LIN {X 0,Y 511.911,Z 787.73,A -85,B 0,C 180,E1 -4052.8,E2 -4052.8} C_VEL
LIN {X 0,Y 511.92,Z 784.945,A -85,B 0,C 180,E1 -4055.058,E2 -4055.058} C_VEL
LIN {X 0,Y 511.96,Z 780.479,A -85,B 0,C 180,E1 -4057.294,E2 -4057.294} C_VEL
LIN {X 0,Y 512.078,Z 774.263,A -85,B 0,C 180,E1 -4059.555,E2 -4059.555} C_VEL
LIN {X 0,Y 512.293,Z 766.172,A -85,B 0,C 180,E1 -4061.827,E2 -4061.827} C_VEL
LIN {X 0,Y 512.637,Z 756.556,A -85,B 0,C 180,E1 -4063.997,E2 -4063.997} C_VEL
LIN {X 0,Y 513.141,Z 745.479,A -85,B 0,C 180,E1 -4066.064,E2 -4066.064} C_VEL
LIN {X 0,Y 513.792,Z 732.943,A -85,B 0,C 180,E1 -4068.025,E2 -4068.025} C_VEL
LIN {X 0,Y 514.601,Z 718.86,A -85,B 0,C 180,E1 -4069.881,E2 -4069.881} C_VEL
LIN {X 0,Y 515.516,Z 703.77,A -85,B 0,C 180,E1 -4071.571,E2 -4071.571} C_VEL
LIN {X 0,Y 516.554,Z 687.043,A -85,B 0,C 180,E1 -4073.158,E2 -4073.158} C_VEL
LIN {X 0,Y 517.654,Z 668.921,A -85,B 0,C 180,E1 -4074.599,E2 -4074.599} C_VEL
LIN {X 0,Y 518.736,Z 650.255,A -85,B 0,C 180,E1 -4075.825,E2 -4075.825} C_VEL
LIN {X 0,Y 519.635,Z 632.605,A -85,B 0,C 180,E1 -4076.772,E2 -4076.772} C_VEL
LIN {X 0,Y 520.342,Z 613.516,A -85,B 0,C 180,E1 -4077.557,E2 -4077.557} C_VEL
LIN {X 0,Y 520.963,Z 593.158,A -85,B 0,C 180,E1 -4078.186,E2 -4078.186} C_VEL
LIN {X 0,Y 521.396,Z 571.634,A -85,B 0,C 180,E1 -4078.64,E2 -4078.64} C_VEL
LIN {X 0,Y 522.992,Z 374.414,A -85,B 0,C 180,E1 -4081.484,E2 -4081.484} C_VEL
LIN {X 0,Y 523.224,Z 329.363,A -85,B 0,C 180,E1 -4082.176,E2 -4082.176} C_VEL
LIN {X 0,Y 521.156,Z 316.493,A -85,B 0,C 180,E1 -4082.526,E2 -4082.526} C_VEL
LIN {X 0,Y 521.816,Z 297.274,A -85,B 0,C 180,E1 -4083.935,E2 -4083.935} C_VEL
LIN {X 0,Y 514.978,Z 278.961,A -85,B 0,C 180,E1 -4085.941,E2 -4085.941} C_VEL
LIN {X 0,Y 512.679,Z 272.854,A -85,B 0,C 180,E1 -4086.732,E2 -4086.732} C_VEL
LIN {X 0,Y 512.623,Z 272.631,A -85,B 0,C 180,E1 -4090.13,E2 -4090.13} C_VEL
LIN {X 0,Y 512.61,Z 272.633,A -85,B 0,C 180,E1 -4093.67,E2 -4093.67} C_VEL
LIN {X 0,Y 512.639,Z 272.631,A -85,B 0,C 180,E1 -4097.102,E2 -4097.102} C_VEL
LIN {X 0,Y 512.649,Z 272.63,A -85,B 0,C 180,E1 -4100.566,E2 -4100.566} C_VEL
LIN {X 0,Y 512.604,Z 272.635,A -85,B 0,C 180,E1 -4103.91,E2 -4103.91} C_VEL
LIN {X 0,Y 512.644,Z 272.869,A -85,B 0,C 180,E1 -4105.454,E2 -4105.454} C_VEL
LIN {X 0,Y 516.614,Z 283.424,A -85,B 0,C 180,E1 -4106.934,E2 -4106.934} C_VEL
LIN {X 0,Y 520.776,Z 295.802,A -85,B 0,C 180,E1 -4108.454,E2 -4108.454} C_VEL
LIN {X 0,Y 518.7,Z 337.157,A -85,B 0,C 180,E1 -4112.069,E2 -4112.069} C_VEL
LIN {X 0,Y 518.616,Z 342.587,A -85,B 0,C 180,E1 -4112.489,E2 -4112.489} C_VEL
LIN {X 0,Y 520.868,Z 357.617,A -85,B 0,C 180,E1 -4112.895,E2 -4112.895} C_VEL
LIN {X 0,Y 518.908,Z 559.958,A -85,B 0,C 180,E1 -4115.886,E2 -4115.886} C_VEL
LIN {X 0,Y 518.407,Z 579.62,A -85,B 0,C 180,E1 -4116.386,E2 -4116.386} C_VEL
LIN {X 0,Y 517.798,Z 597.604,A -85,B 0,C 180,E1 -4117.042,E2 -4117.042} C_VEL
LIN {X 0,Y 517.068,Z 615.514,A -85,B 0,C 180,E1 -4117.908,E2 -4117.908} C_VEL
LIN {X 0,Y 516.22,Z 633.368,A -85,B 0,C 180,E1 -4119.003,E2 -4119.003} C_VEL
LIN {X 0,Y 515.38,Z 650.152,A -85,B 0,C 180,E1 -4120.272,E2 -4120.272} C_VEL
LIN {X 0,Y 514.552,Z 665.731,A -85,B 0,C 180,E1 -4121.711,E2 -4121.711} C_VEL
LIN {X 0,Y 513.83,Z 679.746,A -85,B 0,C 180,E1 -4123.263,E2 -4123.263} C_VEL
LIN {X 0,Y 513.204,Z 692.76,A -85,B 0,C 180,E1 -4124.983,E2 -4124.983} C_VEL
LIN {X 0,Y 512.71,Z 704.206,A -85,B 0,C 180,E1 -4126.811,E2 -4126.811} C_VEL
LIN {X 0,Y 512.352,Z 714.139,A -85,B 0,C 180,E1 -4128.747,E2 -4128.747} C_VEL
LIN {X 0,Y 512.116,Z 722.573,A -85,B 0,C 180,E1 -4130.788,E2 -4130.788} C_VEL
LIN {X 0,Y 511.992,Z 729.132,A -85,B 0,C 180,E1 -4132.821,E2 -4132.821} C_VEL
LIN {X 0,Y 511.937,Z 734.158,A -85,B 0,C 180,E1 -4134.958,E2 -4134.958} C_VEL
LIN {X 0,Y 511.914,Z 737.334,A -85,B 0,C 180,E1 -4137.09,E2 -4137.09} C_VEL
LIN {X 0,Y 511.917,Z 738.827,A -85,B 0,C 180,E1 -4139.217,E2 -4139.217} C_VEL
LIN {X 0,Y 511.911,Z 738.673,A -85,B 0,C 180,E1 -4141.343,E2 -4141.343} C_VEL
LIN {X 0,Y 511.912,Z 736.707,A -85,B 0,C 180,E1 -4143.547,E2 -4143.547} C_VEL
LIN {X 0,Y 511.942,Z 732.933,A -85,B 0,C 180,E1 -4145.717,E2 -4145.717} C_VEL
LIN {X 0,Y 512.015,Z 727.399,A -85,B 0,C 180,E1 -4147.857,E2 -4147.857} C_VEL
LIN {X 0,Y 512.174,Z 720.364,A -85,B 0,C 180,E1 -4149.892,E2 -4149.892} C_VEL
LIN {X 0,Y 512.432,Z 711.904,A -85,B 0,C 180,E1 -4151.823,E2 -4151.823} C_VEL
LIN {X 0,Y 512.822,Z 701.375,A -85,B 0,C 180,E1 -4153.761,E2 -4153.761} C_VEL
LIN {X 0,Y 513.355,Z 689.287,A -85,B 0,C 180,E1 -4155.592,E2 -4155.592} C_VEL
LIN {X 0,Y 514.033,Z 675.591,A -85,B 0,C 180,E1 -4157.314,E2 -4157.314} C_VEL
LIN {X 0,Y 514.776,Z 661.344,A -85,B 0,C 180,E1 -4158.81,E2 -4158.81} C_VEL
LIN {X 0,Y 515.609,Z 645.529,A -85,B 0,C 180,E1 -4160.193,E2 -4160.193} C_VEL
LIN {X 0,Y 516.449,Z 628.721,A -85,B 0,C 180,E1 -4161.398,E2 -4161.398} C_VEL
LIN {X 0,Y 517.278,Z 610.536,A -85,B 0,C 180,E1 -4162.443,E2 -4162.443} C_VEL
LIN {X 0,Y 518.022,Z 591.934,A -85,B 0,C 180,E1 -4163.277,E2 -4163.277} C_VEL
LIN {X 0,Y 518.599,Z 572.89,A -85,B 0,C 180,E1 -4163.901,E2 -4163.901} C_VEL
LIN {X 0,Y 519.014,Z 553.054,A -85,B 0,C 180,E1 -4164.326,E2 -4164.326} C_VEL
LIN {X 0,Y 520.123,Z 426.027,A -85,B 0,C 180,E1 -4166.177,E2 -4166.177} C_VEL
LIN {X 0,Y 519.314,Z 418.442,A -85,B 0,C 180,E1 -4166.337,E2 -4166.337} C_VEL
LIN {X 0,Y 513.976,Z 398.623,A -85,B 0,C 180,E1 -4166.947,E2 -4166.947} C_VEL
LIN {X 0,Y 513.364,Z 392.104,A -85,B 0,C 180,E1 -4167.084,E2 -4167.084} C_VEL
LIN {X 0,Y 513.545,Z 356.301,A -85,B 0,C 180,E1 -4167.633,E2 -4167.633} C_VEL
LIN {X 0,Y 511.161,Z 341.819,A -85,B 0,C 180,E1 -4168.047,E2 -4168.047} C_VEL
LIN {X 0,Y 513.119,Z 299.865,A -85,B 0,C 180,E1 -4171.679,E2 -4171.679} C_VEL
LIN {X 0,Y 513.068,Z 297.719,A -85,B 0,C 180,E1 -4171.879,E2 -4171.879} C_VEL
LIN {X 0,Y 506.338,Z 278.626,A -85,B 0,C 180,E1 -4174.167,E2 -4174.167} C_VEL
LIN {X 0,Y 504.722,Z 273.804,A -85,B 0,C 180,E1 -4174.805,E2 -4174.805} C_VEL
LIN {X 0,Y 504.673,Z 273.62,A -85,B 0,C 180,E1 -4178.181,E2 -4178.181} C_VEL
LIN {X 0,Y 504.694,Z 273.612,A -85,B 0,C 180,E1 -4181.678,E2 -4181.678} C_VEL
LIN {X 0,Y 504.706,Z 273.617,A -85,B 0,C 180,E1 -4185.173,E2 -4185.173} C_VEL
LIN {X 0,Y 504.71,Z 273.619,A -85,B 0,C 180,E1 -4188.723,E2 -4188.723} C_VEL
LIN {X 0,Y 504.699,Z 273.618,A -85,B 0,C 180,E1 -4192.253,E2 -4192.253} C_VEL
LIN {X 0,Y 504.707,Z 273.613,A -85,B 0,C 180,E1 -4195.762,E2 -4195.762} C_VEL
LIN {X 0,Y 504.69,Z 273.612,A -85,B 0,C 180,E1 -4199.297,E2 -4199.297} C_VEL
LIN {X 0,Y 504.681,Z 273.619,A -85,B 0,C 180,E1 -4202.817,E2 -4202.817} C_VEL
LIN {X 0,Y 504.705,Z 273.616,A -85,B 0,C 180,E1 -4206.286,E2 -4206.286} C_VEL
LIN {X 0,Y 504.708,Z 273.614,A -85,B 0,C 180,E1 -4209.835,E2 -4209.835} C_VEL
LIN {X 0,Y 504.659,Z 273.622,A -85,B 0,C 180,E1 -4213.185,E2 -4213.185} C_VEL
LIN {X 0,Y 504.648,Z 273.601,A -85,B 0,C 180,E1 -4216.712,E2 -4216.712} C_VEL
LIN {X 0,Y 504.657,Z 273.717,A -85,B 0,C 180,E1 -4219.208,E2 -4219.208} C_VEL
LIN {X 0,Y 505.095,Z 275.399,A -85,B 0,C 180,E1 -4219.448,E2 -4219.448} C_VEL
LIN {X 0,Y 511.329,Z 294.509,A -85,B 0,C 180,E1 -4221.424,E2 -4221.424} C_VEL
LIN {X 0,Y 510.714,Z 334.383,A -85,B 0,C 180,E1 -4224.663,E2 -4224.663} C_VEL
LIN {X 0,Y 509.833,Z 376.612,A -85,B 0,C 180,E1 -4228.088,E2 -4228.088} C_VEL
LIN {X 0,Y 508.721,Z 421.729,A -85,B 0,C 180,E1 -4231.744,E2 -4231.744} C_VEL
LIN {X 0,Y 507.706,Z 464.389,A -85,B 0,C 180,E1 -4235.196,E2 -4235.196} C_VEL
LIN {X 0,Y 507.513,Z 474.435,A -85,B 0,C 180,E1 -4235.982,E2 -4235.982} C_VEL
LIN {X 0,Y 508.534,Z 485.17,A -85,B 0,C 180,E1 -4236.182,E2 -4236.182} C_VEL
LIN {X 0,Y 507.591,Z 616.922,A -85,B 0,C 180,E1 -4238.102,E2 -4238.102} C_VEL
LIN {X 0,Y 507.323,Z 632.874,A -85,B 0,C 180,E1 -4238.542,E2 -4238.542} C_VEL
LIN {X 0,Y 506.925,Z 648.572,A -85,B 0,C 180,E1 -4239.192,E2 -4239.192} C_VEL
LIN {X 0,Y 506.455,Z 663.014,A -85,B 0,C 180,E1 -4240.003,E2 -4240.003} C_VEL
LIN {X 0,Y 505.905,Z 677.326,A -85,B 0,C 180,E1 -4241.051,E2 -4241.051} C_VEL
LIN {X 0,Y 505.414,Z 690.119,A -85,B 0,C 180,E1 -4242.234,E2 -4242.234} C_VEL
LIN {X 0,Y 504.93,Z 702.107,A -85,B 0,C 180,E1 -4243.628,E2 -4243.628} C_VEL
LIN {X 0,Y 504.569,Z 711.921,A -85,B 0,C 180,E1 -4245.044,E2 -4245.044} C_VEL
LIN {X 0,Y 504.268,Z 721.08,A -85,B 0,C 180,E1 -4246.724,E2 -4246.724} C_VEL
LIN {X 0,Y 504.091,Z 728.094,A -85,B 0,C 180,E1 -4248.382,E2 -4248.382} C_VEL
LIN {X 0,Y 503.989,Z 733.734,A -85,B 0,C 180,E1 -4250.217,E2 -4250.217} C_VEL
LIN {X 0,Y 503.95,Z 737.461,A -85,B 0,C 180,E1 -4252.022,E2 -4252.022} C_VEL
LIN {X 0,Y 503.935,Z 739.424,A -85,B 0,C 180,E1 -4253.874,E2 -4253.874} C_VEL
LIN {X 0,Y 503.935,Z 739.676,A -85,B 0,C 180,E1 -4255.753,E2 -4255.753} C_VEL
LIN {X 0,Y 503.943,Z 738.029,A -85,B 0,C 180,E1 -4257.661,E2 -4257.661} C_VEL
LIN {X 0,Y 503.976,Z 734.754,A -85,B 0,C 180,E1 -4259.471,E2 -4259.471} C_VEL
LIN {X 0,Y 504.057,Z 729.721,A -85,B 0,C 180,E1 -4261.246,E2 -4261.246} C_VEL
LIN {X 0,Y 504.23,Z 722.652,A -85,B 0,C 180,E1 -4263.044,E2 -4263.044} C_VEL
LIN {X 0,Y 504.492,Z 714.234,A -85,B 0,C 180,E1 -4264.665,E2 -4264.665} C_VEL
LIN {X 0,Y 504.853,Z 704.388,A -85,B 0,C 180,E1 -4266.168,E2 -4266.168} C_VEL
LIN {X 0,Y 505.3,Z 693.074,A -85,B 0,C 180,E1 -4267.548,E2 -4267.548} C_VEL
LIN {X 0,Y 505.831,Z 679.711,A -85,B 0,C 180,E1 -4268.848,E2 -4268.848} C_VEL
LIN {X 0,Y 506.327,Z 666.781,A -85,B 0,C 180,E1 -4269.842,E2 -4269.842} C_VEL
LIN {X 0,Y 506.852,Z 651.387,A -85,B 0,C 180,E1 -4270.763,E2 -4270.763} C_VEL
LIN {X 0,Y 507.266,Z 635.918,A -85,B 0,C 180,E1 -4271.442,E2 -4271.442} C_VEL
LIN {X 0,Y 507.556,Z 619.27,A -85,B 0,C 180,E1 -4271.94,E2 -4271.94} C_VEL
LIN {X 0,Y 507.753,Z 593.359,A -85,B 0,C 180,E1 -4272.356,E2 -4272.356} C_VEL
LIN {X 0,Y 508.34,Z 481.293,A -85,B 0,C 180,E1 -4273.974,E2 -4273.974} C_VEL
LIN {X 0,Y 507.457,Z 474.005,A -85,B 0,C 180,E1 -4274.135,E2 -4274.135} C_VEL
LIN {X 0,Y 508.502,Z 429.195,A -85,B 0,C 180,E1 -4277.741,E2 -4277.741} C_VEL
LIN {X 0,Y 509.471,Z 389.356,A -85,B 0,C 180,E1 -4280.951,E2 -4280.951} C_VEL
LIN {X 0,Y 510.24,Z 346.659,A -85,B 0,C 180,E1 -4284.346,E2 -4284.346} C_VEL
LIN {X 0,Y 510.701,Z 309.068,A -85,B 0,C 180,E1 -4287.334,E2 -4287.334} C_VEL
LIN {X 0,Y 510.741,Z 292.979,A -85,B 0,C 180,E1 -4288.618,E2 -4288.618} C_VEL
LIN {X 0,Y 504.771,Z 274.004,A -85,B 0,C 180,E1 -4290.512,E2 -4290.512} C_VEL
LIN {X 0,Y 504.69,Z 273.619,A -85,B 0,C 180,E1 -4290.885,E2 -4290.885} C_VEL
LIN {X 0,Y 504.709,Z 273.616,A -85,B 0,C 180,E1 -4294.336,E2 -4294.336} C_VEL
LIN {X 0,Y 504.669,Z 273.622,A -85,B 0,C 180,E1 -4297.764,E2 -4297.764} C_VEL
LIN {X 0,Y 504.671,Z 273.614,A -85,B 0,C 180,E1 -4301.279,E2 -4301.279} C_VEL
LIN {X 0,Y 504.711,Z 273.613,A -85,B 0,C 180,E1 -4304.739,E2 -4304.739} C_VEL
LIN {X 0,Y 504.694,Z 273.622,A -85,B 0,C 180,E1 -4308.225,E2 -4308.225} C_VEL
LIN {X 0,Y 504.667,Z 273.617,A -85,B 0,C 180,E1 -4311.684,E2 -4311.684} C_VEL
LIN {X 0,Y 504.687,Z 273.615,A -85,B 0,C 180,E1 -4315.192,E2 -4315.192} C_VEL
LIN {X 0,Y 504.711,Z 273.617,A -85,B 0,C 180,E1 -4318.637,E2 -4318.637} C_VEL
LIN {X 0,Y 504.675,Z 273.618,A -85,B 0,C 180,E1 -4322.043,E2 -4322.043} C_VEL
LIN {X 0,Y 504.673,Z 273.617,A -85,B 0,C 180,E1 -4325.571,E2 -4325.571} C_VEL
LIN {X 0,Y 504.709,Z 273.612,A -85,B 0,C 180,E1 -4329.004,E2 -4329.004} C_VEL
LIN {X 0,Y 504.704,Z 273.617,A -85,B 0,C 180,E1 -4332.586,E2 -4332.586} C_VEL
LIN {X 0,Y 504.673,Z 273.615,A -85,B 0,C 180,E1 -4335.985,E2 -4335.985} C_VEL
LIN {X 0,Y 504.69,Z 273.614,A -85,B 0,C 180,E1 -4339.441,E2 -4339.441} C_VEL
LIN {X 0,Y 504.712,Z 273.617,A -85,B 0,C 180,E1 -4342.971,E2 -4342.971} C_VEL
LIN {X 0,Y 504.691,Z 273.62,A -85,B 0,C 180,E1 -4346.471,E2 -4346.471} C_VEL
LIN {X 0,Y 504.676,Z 273.615,A -85,B 0,C 180,E1 -4349.951,E2 -4349.951} C_VEL
LIN {X 0,Y 504.704,Z 273.613,A -85,B 0,C 180,E1 -4353.417,E2 -4353.417} C_VEL
LIN {X 0,Y 504.708,Z 273.62,A -85,B 0,C 180,E1 -4356.888,E2 -4356.888} C_VEL
LIN {X 0,Y 504.68,Z 273.619,A -85,B 0,C 180,E1 -4360.379,E2 -4360.379} C_VEL
LIN {X 0,Y 504.684,Z 273.618,A -85,B 0,C 180,E1 -4363.9,E2 -4363.9} C_VEL
LIN {X 0,Y 504.71,Z 273.617,A -85,B 0,C 180,E1 -4367.352,E2 -4367.352} C_VEL
LIN {X 0,Y 504.713,Z 273.617,A -85,B 0,C 180,E1 -4370.954,E2 -4370.954} C_VEL
LIN {X 0,Y 504.722,Z 273.854,A -85,B 0,C 180,E1 -4372.645,E2 -4372.645} C_VEL
LIN {X 0,Y 507.634,Z 281.444,A -85,B 0,C 180,E1 -4373.571,E2 -4373.571} C_VEL
LIN {X 0,Y 515.207,Z 300.924,A -85,B 0,C 180,E1 -4375.719,E2 -4375.719} C_VEL
LIN {X 0,Y 514.589,Z 316.443,A -85,B 0,C 180,E1 -4376.864,E2 -4376.864} C_VEL
LIN {X 0,Y 517.105,Z 333.218,A -85,B 0,C 180,E1 -4377.321,E2 -4377.321} C_VEL
LIN {X 0,Y 514.727,Z 530.291,A -85,B 0,C 180,E1 -4380.332,E2 -4380.332} C_VEL
LIN {X 0,Y 514.183,Z 578.441,A -85,B 0,C 180,E1 -4381.071,E2 -4381.071} C_VEL
LIN {X 0,Y 513.538,Z 599.827,A -85,B 0,C 180,E1 -4381.608,E2 -4381.608} C_VEL
LIN {X 0,Y 512.738,Z 620.455,A -85,B 0,C 180,E1 -4382.349,E2 -4382.349} C_VEL
LIN {X 0,Y 511.825,Z 639.514,A -85,B 0,C 180,E1 -4383.24,E2 -4383.24} C_VEL
LIN {X 0,Y 510.774,Z 658.935,A -85,B 0,C 180,E1 -4384.368,E2 -4384.368} C_VEL
LIN {X 0,Y 509.701,Z 677.368,A -85,B 0,C 180,E1 -4385.674,E2 -4385.674} C_VEL
LIN {X 0,Y 508.649,Z 693.186,A -85,B 0,C 180,E1 -4387.035,E2 -4387.035} C_VEL
LIN {X 0,Y 507.519,Z 709.709,A -85,B 0,C 180,E1 -4388.725,E2 -4388.725} C_VEL
LIN {X 0,Y 506.541,Z 724.454,A -85,B 0,C 180,E1 -4390.515,E2 -4390.515} C_VEL
LIN {X 0,Y 505.731,Z 737.586,A -85,B 0,C 180,E1 -4392.394,E2 -4392.394} C_VEL
LIN {X 0,Y 505.077,Z 749.383,A -85,B 0,C 180,E1 -4394.383,E2 -4394.383} C_VEL
LIN {X 0,Y 504.568,Z 760.338,A -85,B 0,C 180,E1 -4396.596,E2 -4396.596} C_VEL
LIN {X 0,Y 504.236,Z 769.256,A -85,B 0,C 180,E1 -4398.796,E2 -4398.796} C_VEL
LIN {X 0,Y 504.048,Z 776.587,A -85,B 0,C 180,E1 -4401.062,E2 -4401.062} C_VEL
LIN {X 0,Y 503.957,Z 782.261,A -85,B 0,C 180,E1 -4403.394,E2 -4403.394} C_VEL
LIN {X 0,Y 503.916,Z 786.089,A -85,B 0,C 180,E1 -4405.677,E2 -4405.677} C_VEL
LIN {X 0,Y 503.911,Z 788.374,A -85,B 0,C 180,E1 -4408.068,E2 -4408.068} C_VEL
LIN {X 0,Y 503.9,Z 788.917,A -85,B 0,C 180,E1 -4410.456,E2 -4410.456} C_VEL
LIN {X 0,Y 503.911,Z 787.842,A -85,B 0,C 180,E1 -4412.731,E2 -4412.731} C_VEL
LIN {X 0,Y 503.922,Z 785.126,A -85,B 0,C 180,E1 -4415.01,E2 -4415.01} C_VEL
LIN {X 0,Y 503.964,Z 780.733,A -85,B 0,C 180,E1 -4417.296,E2 -4417.296} C_VEL
LIN {X 0,Y 504.091,Z 774.616,A -85,B 0,C 180,E1 -4419.592,E2 -4419.592} C_VEL
LIN {X 0,Y 504.314,Z 767.088,A -85,B 0,C 180,E1 -4421.784,E2 -4421.784} C_VEL
LIN {X 0,Y 504.683,Z 757.701,A -85,B 0,C 180,E1 -4423.988,E2 -4423.988} C_VEL
LIN {X 0,Y 505.219,Z 746.825,A -85,B 0,C 180,E1 -4426.086,E2 -4426.086} C_VEL
LIN {X 0,Y 505.915,Z 734.462,A -85,B 0,C 180,E1 -4428.082,E2 -4428.082} C_VEL
LIN {X 0,Y 506.779,Z 720.73,A -85,B 0,C 180,E1 -4429.959,E2 -4429.959} C_VEL
LIN {X 0,Y 507.8,Z 705.486,A -85,B 0,C 180,E1 -4431.727,E2 -4431.727} C_VEL
LIN {X 0,Y 508.908,Z 689.266,A -85,B 0,C 180,E1 -4433.322,E2 -4433.322} C_VEL
LIN {X 0,Y 509.9,Z 674.301,A -85,B 0,C 180,E1 -4434.565,E2 -4434.565} C_VEL
LIN {X 0,Y 510.85,Z 656.652,A -85,B 0,C 180,E1 -4435.755,E2 -4435.755} C_VEL
LIN {X 0,Y 511.789,Z 637.288,A -85,B 0,C 180,E1 -4436.828,E2 -4436.828} C_VEL
LIN {X 0,Y 512.652,Z 616.924,A -85,B 0,C 180,E1 -4437.722,E2 -4437.722} C_VEL
LIN {X 0,Y 513.334,Z 596.303,A -85,B 0,C 180,E1 -4438.406,E2 -4438.406} C_VEL
LIN {X 0,Y 513.865,Z 575.457,A -85,B 0,C 180,E1 -4438.888,E2 -4438.888} C_VEL
LIN {X 0,Y 515.691,Z 379.054,A -85,B 0,C 180,E1 -4441.79,E2 -4441.79} C_VEL
LIN {X 0,Y 516.094,Z 330.597,A -85,B 0,C 180,E1 -4442.562,E2 -4442.562} C_VEL
LIN {X 0,Y 513.987,Z 317.144,A -85,B 0,C 180,E1 -4442.938,E2 -4442.938} C_VEL
LIN {X 0,Y 514.567,Z 300.018,A -85,B 0,C 180,E1 -4444.23,E2 -4444.23} C_VEL
LIN {X 0,Y 508.155,Z 282.576,A -85,B 0,C 180,E1 -4446.223,E2 -4446.223} C_VEL
LIN {X 0,Y 504.746,Z 274.031,A -85,B 0,C 180,E1 -4447.376,E2 -4447.376} C_VEL
LIN {X 0,Y 504.688,Z 273.622,A -85,B 0,C 180,E1 -4448.139,E2 -4448.139} C_VEL
LIN {X 0,Y 504.673,Z 273.623,A -85,B 0,C 180,E1 -4451.677,E2 -4451.677} C_VEL
LIN {X 0,Y 504.696,Z 273.622,A -85,B 0,C 180,E1 -4455.174,E2 -4455.174} C_VEL
LIN {X 0,Y 504.715,Z 273.618,A -85,B 0,C 180,E1 -4458.724,E2 -4458.724} C_VEL
LIN {X 0,Y 504.672,Z 273.622,A -85,B 0,C 180,E1 -4462.108,E2 -4462.108} C_VEL
LIN {X 0,Y 504.745,Z 273.87,A -85,B 0,C 180,E1 -4464.73,E2 -4464.73} C_VEL
LIN {X 0,Y 509.029,Z 284.919,A -85,B 0,C 180,E1 -4466.393,E2 -4466.393} C_VEL
LIN {X 0,Y 513.704,Z 298.842,A -85,B 0,C 180,E1 -4468.182,E2 -4468.182} C_VEL
LIN {X 0,Y 511.459,Z 339.199,A -85,B 0,C 180,E1 -4471.765,E2 -4471.765} C_VEL
LIN {X 0,Y 511.524,Z 342.462,A -85,B 0,C 180,E1 -4471.987,E2 -4471.987} C_VEL
LIN {X 0,Y 513.978,Z 358.746,A -85,B 0,C 180,E1 -4472.456,E2 -4472.456} C_VEL
LIN {X 0,Y 512.461,Z 472.725,A -85,B 0,C 180,E1 -4474.213,E2 -4474.213} C_VEL
LIN {X 0,Y 511.596,Z 560.324,A -85,B 0,C 180,E1 -4475.528,E2 -4475.528} C_VEL
LIN {X 0,Y 511.05,Z 580.056,A -85,B 0,C 180,E1 -4476.039,E2 -4476.039} C_VEL
LIN {X 0,Y 510.37,Z 598.506,A -85,B 0,C 180,E1 -4476.727,E2 -4476.727} C_VEL
LIN {X 0,Y 509.549,Z 616.547,A -85,B 0,C 180,E1 -4477.625,E2 -4477.625} C_VEL
LIN {X 0,Y 508.634,Z 634.223,A -85,B 0,C 180,E1 -4478.735,E2 -4478.735} C_VEL
LIN {X 0,Y 507.715,Z 650.838,A -85,B 0,C 180,E1 -4480.021,E2 -4480.021} C_VEL
LIN {X 0,Y 506.811,Z 666.298,A -85,B 0,C 180,E1 -4481.481,E2 -4481.481} C_VEL
LIN {X 0,Y 505.995,Z 680.673,A -85,B 0,C 180,E1 -4483.114,E2 -4483.114} C_VEL
LIN {X 0,Y 505.316,Z 693.54,A -85,B 0,C 180,E1 -4484.86,E2 -4484.86} C_VEL
LIN {X 0,Y 504.78,Z 704.869,A -85,B 0,C 180,E1 -4486.717,E2 -4486.717} C_VEL
LIN {X 0,Y 504.389,Z 714.671,A -85,B 0,C 180,E1 -4488.683,E2 -4488.683} C_VEL
LIN {X 0,Y 504.132,Z 722.981,A -85,B 0,C 180,E1 -4490.756,E2 -4490.756} C_VEL
LIN {X 0,Y 503.996,Z 729.437,A -85,B 0,C 180,E1 -4492.821,E2 -4492.821} C_VEL
LIN {X 0,Y 503.938,Z 734.369,A -85,B 0,C 180,E1 -4494.992,E2 -4494.992} C_VEL
LIN {X 0,Y 503.913,Z 737.461,A -85,B 0,C 180,E1 -4497.157,E2 -4497.157} C_VEL
LIN {X 0,Y 503.914,Z 738.851,A -85,B 0,C 180,E1 -4499.318,E2 -4499.318} C_VEL
LIN {X 0,Y 503.911,Z 738.608,A -85,B 0,C 180,E1 -4501.478,E2 -4501.478} C_VEL
LIN {X 0,Y 503.912,Z 736.66,A -85,B 0,C 180,E1 -4503.641,E2 -4503.641} C_VEL
LIN {X 0,Y 503.945,Z 732.928,A -85,B 0,C 180,E1 -4505.808,E2 -4505.808} C_VEL
LIN {X 0,Y 504.03,Z 727.395,A -85,B 0,C 180,E1 -4507.982,E2 -4507.982} C_VEL
LIN {X 0,Y 504.204,Z 720.361,A -85,B 0,C 180,E1 -4510.05,E2 -4510.05} C_VEL
LIN {X 0,Y 504.494,Z 711.898,A -85,B 0,C 180,E1 -4512.011,E2 -4512.011} C_VEL
LIN {X 0,Y 504.931,Z 701.366,A -85,B 0,C 180,E1 -4513.98,E2 -4513.98} C_VEL
LIN {X 0,Y 505.526,Z 689.278,A -85,B 0,C 180,E1 -4515.84,E2 -4515.84} C_VEL
LIN {X 0,Y 506.277,Z 675.582,A -85,B 0,C 180,E1 -4517.588,E2 -4517.588} C_VEL
LIN {X 0,Y 507.096,Z 661.337,A -85,B 0,C 180,E1 -4519.106,E2 -4519.106} C_VEL
LIN {X 0,Y 508.011,Z 645.517,A -85,B 0,C 180,E1 -4520.508,E2 -4520.508} C_VEL
LIN {X 0,Y 508.934,Z 628.612,A -85,B 0,C 180,E1 -4521.736,E2 -4521.736} C_VEL
LIN {X 0,Y 509.832,Z 610.521,A -85,B 0,C 180,E1 -4522.789,E2 -4522.789} C_VEL
LIN {X 0,Y 510.615,Z 592.575,A -85,B 0,C 180,E1 -4523.606,E2 -4523.606} C_VEL
LIN {X 0,Y 511.25,Z 573.74,A -85,B 0,C 180,E1 -4524.242,E2 -4524.242} C_VEL
LIN {X 0,Y 511.696,Z 554.425,A -85,B 0,C 180,E1 -4524.671,E2 -4524.671} C_VEL
LIN {X 0,Y 513.364,Z 392.104,A -85,B 0,C 180,E1 -4527.084,E2 -4527.084} C_VEL
LIN {X 0,Y 512.593,Z 383.441,A -85,B 0,C 180,E1 -4527.264,E2 -4527.264} C_VEL
LIN {X 0,Y 506.641,Z 358.228,A -85,B 0,C 180,E1 -4528.032,E2 -4528.032} C_VEL
LIN {X 0,Y 503.93,Z 341.479,A -85,B 0,C 180,E1 -4528.53,E2 -4528.53} C_VEL
LIN {X 0,Y 505.986,Z 301.18,A -85,B 0,C 180,E1 -4532.069,E2 -4532.069} C_VEL
LIN {X 0,Y 499.705,Z 283.022,A -85,B 0,C 180,E1 -4534.271,E2 -4534.271} C_VEL
LIN {X 0,Y 496.793,Z 274.791,A -85,B 0,C 180,E1 -4535.362,E2 -4535.362} C_VEL
LIN {X 0,Y 496.772,Z 274.605,A -85,B 0,C 180,E1 -4538.901,E2 -4538.901} C_VEL
LIN {X 0,Y 496.748,Z 274.605,A -85,B 0,C 180,E1 -4542.4,E2 -4542.4} C_VEL
LIN {X 0,Y 496.751,Z 274.607,A -85,B 0,C 180,E1 -4546.018,E2 -4546.018} C_VEL
LIN {X 0,Y 496.769,Z 274.603,A -85,B 0,C 180,E1 -4549.601,E2 -4549.601} C_VEL
LIN {X 0,Y 496.757,Z 274.604,A -85,B 0,C 180,E1 -4553.143,E2 -4553.143} C_VEL
LIN {X 0,Y 496.761,Z 274.607,A -85,B 0,C 180,E1 -4556.667,E2 -4556.667} C_VEL
LIN {X 0,Y 496.769,Z 274.598,A -85,B 0,C 180,E1 -4560.188,E2 -4560.188} C_VEL
LIN {X 0,Y 496.768,Z 274.604,A -85,B 0,C 180,E1 -4563.716,E2 -4563.716} C_VEL
LIN {X 0,Y 496.734,Z 274.607,A -85,B 0,C 180,E1 -4567.206,E2 -4567.206} C_VEL
LIN {X 0,Y 496.727,Z 274.609,A -85,B 0,C 180,E1 -4570.745,E2 -4570.745} C_VEL
LIN {X 0,Y 496.753,Z 274.6,A -85,B 0,C 180,E1 -4574.232,E2 -4574.232} C_VEL
LIN {X 0,Y 496.743,Z 274.605,A -85,B 0,C 180,E1 -4577.68,E2 -4577.68} C_VEL
LIN {X 0,Y 496.744,Z 274.899,A -85,B 0,C 180,E1 -4578.828,E2 -4578.828} C_VEL
LIN {X 0,Y 503.539,Z 295.552,A -85,B 0,C 180,E1 -4581.031,E2 -4581.031} C_VEL
LIN {X 0,Y 503.974,Z 298.794,A -85,B 0,C 180,E1 -4581.327,E2 -4581.327} C_VEL
LIN {X 0,Y 503.208,Z 340.602,A -85,B 0,C 180,E1 -4584.755,E2 -4584.755} C_VEL
LIN {X 0,Y 502.249,Z 380.984,A -85,B 0,C 180,E1 -4588.059,E2 -4588.059} C_VEL
LIN {X 0,Y 501.067,Z 425.768,A -85,B 0,C 180,E1 -4591.714,E2 -4591.714} C_VEL
LIN {X 0,Y 500.006,Z 468.043,A -85,B 0,C 180,E1 -4595.161,E2 -4595.161} C_VEL
LIN {X 0,Y 499.903,Z 474.861,A -85,B 0,C 180,E1 -4595.684,E2 -4595.684} C_VEL
LIN {X 0,Y 500.969,Z 485.924,A -85,B 0,C 180,E1 -4595.895,E2 -4595.895} C_VEL
LIN {X 0,Y 499.941,Z 617.34,A -85,B 0,C 180,E1 -4597.84,E2 -4597.84} C_VEL
LIN {X 0,Y 499.655,Z 633.277,A -85,B 0,C 180,E1 -4598.286,E2 -4598.286} C_VEL
LIN {X 0,Y 499.205,Z 649.81,A -85,B 0,C 180,E1 -4598.987,E2 -4598.987} C_VEL
LIN {X 0,Y 498.696,Z 664.017,A -85,B 0,C 180,E1 -4599.811,E2 -4599.811} C_VEL
LIN {X 0,Y 498.107,Z 678.224,A -85,B 0,C 180,E1 -4600.875,E2 -4600.875} C_VEL
LIN {X 0,Y 497.578,Z 690.76,A -85,B 0,C 180,E1 -4602.061,E2 -4602.061} C_VEL
LIN {X 0,Y 497.048,Z 702.83,A -85,B 0,C 180,E1 -4603.493,E2 -4603.493} C_VEL
LIN {X 0,Y 496.653,Z 712.568,A -85,B 0,C 180,E1 -4604.931,E2 -4604.931} C_VEL
LIN {X 0,Y 496.323,Z 721.598,A -85,B 0,C 180,E1 -4606.621,E2 -4606.621} C_VEL
LIN {X 0,Y 496.123,Z 728.676,A -85,B 0,C 180,E1 -4608.334,E2 -4608.334} C_VEL
LIN {X 0,Y 496.01,Z 734.174,A -85,B 0,C 180,E1 -4610.162,E2 -4610.162} C_VEL
LIN {X 0,Y 495.963,Z 737.914,A -85,B 0,C 180,E1 -4612.021,E2 -4612.021} C_VEL
LIN {X 0,Y 495.946,Z 739.841,A -85,B 0,C 180,E1 -4613.904,E2 -4613.904} C_VEL
LIN {X 0,Y 495.945,Z 740.052,A -85,B 0,C 180,E1 -4615.813,E2 -4615.813} C_VEL
LIN {X 0,Y 495.956,Z 738.355,A -85,B 0,C 180,E1 -4617.754,E2 -4617.754} C_VEL
LIN {X 0,Y 496.004,Z 734.845,A -85,B 0,C 180,E1 -4619.677,E2 -4619.677} C_VEL
LIN {X 0,Y 496.106,Z 729.548,A -85,B 0,C 180,E1 -4621.512,E2 -4621.512} C_VEL
LIN {X 0,Y 496.302,Z 722.599,A -85,B 0,C 180,E1 -4623.272,E2 -4623.272} C_VEL
LIN {X 0,Y 496.624,Z 713.491,A -85,B 0,C 180,E1 -4625.013,E2 -4625.013} C_VEL
LIN {X 0,Y 497.041,Z 703.344,A -85,B 0,C 180,E1 -4626.542,E2 -4626.542} C_VEL
LIN {X 0,Y 497.549,Z 691.637,A -85,B 0,C 180,E1 -4627.944,E2 -4627.944} C_VEL
LIN {X 0,Y 498.077,Z 679.489,A -85,B 0,C 180,E1 -4629.119,E2 -4629.119} C_VEL
LIN {X 0,Y 498.659,Z 665.144,A -85,B 0,C 180,E1 -4630.211,E2 -4630.211} C_VEL
LIN {X 0,Y 499.193,Z 650.674,A -85,B 0,C 180,E1 -4631.067,E2 -4631.067} C_VEL
LIN {X 0,Y 499.631,Z 634.514,A -85,B 0,C 180,E1 -4631.763,E2 -4631.763} C_VEL
LIN {X 0,Y 499.922,Z 618.388,A -85,B 0,C 180,E1 -4632.231,E2 -4632.231} C_VEL
LIN {X 0,Y 500.3,Z 568.29,A -85,B 0,C 180,E1 -4632.995,E2 -4632.995} C_VEL
LIN {X 0,Y 500.781,Z 482.143,A -85,B 0,C 180,E1 -4634.261,E2 -4634.261} C_VEL
LIN {X 0,Y 499.842,Z 474.397,A -85,B 0,C 180,E1 -4634.434,E2 -4634.434} C_VEL
LIN {X 0,Y 500.963,Z 429.094,A -85,B 0,C 180,E1 -4638.11,E2 -4638.11} C_VEL
LIN {X 0,Y 501.829,Z 393.421,A -85,B 0,C 180,E1 -4640.988,E2 -4640.988} C_VEL
LIN {X 0,Y 502.557,Z 361.365,A -85,B 0,C 180,E1 -4643.567,E2 -4643.567} C_VEL
LIN {X 0,Y 503.208,Z 320.138,A -85,B 0,C 180,E1 -4646.878,E2 -4646.878} C_VEL
LIN {X 0,Y 503.4,Z 295.62,A -85,B 0,C 180,E1 -4648.841,E2 -4648.841} C_VEL
LIN {X 0,Y 496.791,Z 274.932,A -85,B 0,C 180,E1 -4650.951,E2 -4650.951} C_VEL
LIN {X 0,Y 496.729,Z 274.611,A -85,B 0,C 180,E1 -4651.637,E2 -4651.637} C_VEL
LIN {X 0,Y 496.731,Z 274.611,A -85,B 0,C 180,E1 -4655.248,E2 -4655.248} C_VEL
LIN {X 0,Y 496.766,Z 274.602,A -85,B 0,C 180,E1 -4658.758,E2 -4658.758} C_VEL
LIN {X 0,Y 496.764,Z 274.605,A -85,B 0,C 180,E1 -4662.306,E2 -4662.306} C_VEL
LIN {X 0,Y 496.729,Z 274.608,A -85,B 0,C 180,E1 -4665.784,E2 -4665.784} C_VEL
LIN {X 0,Y 496.736,Z 274.605,A -85,B 0,C 180,E1 -4669.328,E2 -4669.328} C_VEL
LIN {X 0,Y 496.774,Z 274.603,A -85,B 0,C 180,E1 -4672.852,E2 -4672.852} C_VEL
LIN {X 0,Y 496.764,Z 274.607,A -85,B 0,C 180,E1 -4676.422,E2 -4676.422} C_VEL
LIN {X 0,Y 496.733,Z 274.608,A -85,B 0,C 180,E1 -4679.884,E2 -4679.884} C_VEL
LIN {X 0,Y 496.738,Z 274.604,A -85,B 0,C 180,E1 -4683.462,E2 -4683.462} C_VEL
LIN {X 0,Y 496.773,Z 274.603,A -85,B 0,C 180,E1 -4686.936,E2 -4686.936} C_VEL
LIN {X 0,Y 496.757,Z 274.606,A -85,B 0,C 180,E1 -4690.436,E2 -4690.436} C_VEL
LIN {X 0,Y 496.734,Z 274.606,A -85,B 0,C 180,E1 -4693.977,E2 -4693.977} C_VEL
LIN {X 0,Y 496.744,Z 274.605,A -85,B 0,C 180,E1 -4697.573,E2 -4697.573} C_VEL
LIN {X 0,Y 496.771,Z 274.602,A -85,B 0,C 180,E1 -4701.117,E2 -4701.117} C_VEL
LIN {X 0,Y 496.763,Z 274.607,A -85,B 0,C 180,E1 -4704.622,E2 -4704.622} C_VEL
LIN {X 0,Y 496.738,Z 274.607,A -85,B 0,C 180,E1 -4708.165,E2 -4708.165} C_VEL
LIN {X 0,Y 496.746,Z 274.603,A -85,B 0,C 180,E1 -4711.691,E2 -4711.691} C_VEL
LIN {X 0,Y 496.772,Z 274.604,A -85,B 0,C 180,E1 -4715.202,E2 -4715.202} C_VEL
LIN {X 0,Y 496.767,Z 274.609,A -85,B 0,C 180,E1 -4718.752,E2 -4718.752} C_VEL
LIN {X 0,Y 496.739,Z 274.609,A -85,B 0,C 180,E1 -4722.244,E2 -4722.244} C_VEL
LIN {X 0,Y 496.751,Z 274.605,A -85,B 0,C 180,E1 -4725.77,E2 -4725.77} C_VEL
LIN {X 0,Y 496.772,Z 274.607,A -85,B 0,C 180,E1 -4729.301,E2 -4729.301} C_VEL
LIN {X 0,Y 496.777,Z 274.865,A -85,B 0,C 180,E1 -4732.056,E2 -4732.056} C_VEL
LIN {X 0,Y 500.523,Z 284.291,A -85,B 0,C 180,E1 -4733.23,E2 -4733.23} C_VEL
LIN {X 0,Y 508.094,Z 303.988,A -85,B 0,C 180,E1 -4735.441,E2 -4735.441} C_VEL
LIN {X 0,Y 507.57,Z 316.675,A -85,B 0,C 180,E1 -4736.384,E2 -4736.384} C_VEL
LIN {X 0,Y 510.176,Z 334.45,A -85,B 0,C 180,E1 -4736.888,E2 -4736.888} C_VEL
LIN {X 0,Y 508.469,Z 453.813,A -85,B 0,C 180,E1 -4738.763,E2 -4738.763} C_VEL
LIN {X 0,Y 506.934,Z 577.933,A -85,B 0,C 180,E1 -4740.68,E2 -4740.68} C_VEL
LIN {X 0,Y 506.225,Z 599.572,A -85,B 0,C 180,E1 -4741.231,E2 -4741.231} C_VEL
LIN {X 0,Y 505.38,Z 619.891,A -85,B 0,C 180,E1 -4741.969,E2 -4741.969} C_VEL
LIN {X 0,Y 504.378,Z 639.254,A -85,B 0,C 180,E1 -4742.883,E2 -4742.883} C_VEL
LIN {X 0,Y 503.262,Z 658.557,A -85,B 0,C 180,E1 -4744.019,E2 -4744.019} C_VEL
LIN {X 0,Y 502.09,Z 677.202,A -85,B 0,C 180,E1 -4745.359,E2 -4745.359} C_VEL
LIN {X 0,Y 500.925,Z 694.485,A -85,B 0,C 180,E1 -4746.847,E2 -4746.847} C_VEL
LIN {X 0,Y 499.847,Z 710.302,A -85,B 0,C 180,E1 -4748.458,E2 -4748.458} C_VEL
LIN {X 0,Y 498.832,Z 724.453,A -85,B 0,C 180,E1 -4750.201,E2 -4750.201} C_VEL
LIN {X 0,Y 497.924,Z 737.789,A -85,B 0,C 180,E1 -4752.141,E2 -4752.141} C_VEL
LIN {X 0,Y 497.213,Z 749.382,A -85,B 0,C 180,E1 -4754.13,E2 -4754.13} C_VEL
LIN {X 0,Y 496.65,Z 760.337,A -85,B 0,C 180,E1 -4756.378,E2 -4756.378} C_VEL
LIN {X 0,Y 496.279,Z 769.255,A -85,B 0,C 180,E1 -4758.614,E2 -4758.614} C_VEL
LIN {X 0,Y 496.067,Z 776.378,A -85,B 0,C 180,E1 -4760.839,E2 -4760.839} C_VEL
LIN {X 0,Y 495.965,Z 782.008,A -85,B 0,C 180,E1 -4763.17,E2 -4763.17} C_VEL
LIN {X 0,Y 495.918,Z 785.929,A -85,B 0,C 180,E1 -4765.491,E2 -4765.491} C_VEL
LIN {X 0,Y 495.911,Z 788.305,A -85,B 0,C 180,E1 -4767.921,E2 -4767.921} C_VEL
LIN {X 0,Y 495.906,Z 788.962,A -85,B 0,C 180,E1 -4770.232,E2 -4770.232} C_VEL
LIN {X 0,Y 495.908,Z 788.03,A -85,B 0,C 180,E1 -4772.544,E2 -4772.544} C_VEL
LIN {X 0,Y 495.924,Z 785.445,A -85,B 0,C 180,E1 -4774.859,E2 -4774.859} C_VEL
LIN {X 0,Y 495.964,Z 781.241,A -85,B 0,C 180,E1 -4777.181,E2 -4777.181} C_VEL
LIN {X 0,Y 496.095,Z 775.322,A -85,B 0,C 180,E1 -4779.514,E2 -4779.514} C_VEL
LIN {X 0,Y 496.335,Z 767.956,A -85,B 0,C 180,E1 -4781.753,E2 -4781.753} C_VEL
LIN {X 0,Y 496.733,Z 758.589,A -85,B 0,C 180,E1 -4784.023,E2 -4784.023} C_VEL
LIN {X 0,Y 497.288,Z 748.099,A -85,B 0,C 180,E1 -4786.11,E2 -4786.11} C_VEL
LIN {X 0,Y 498.033,Z 736.03,A -85,B 0,C 180,E1 -4788.131,E2 -4788.131} C_VEL
LIN {X 0,Y 499.023,Z 721.655,A -85,B 0,C 180,E1 -4790.16,E2 -4790.16} C_VEL
LIN {X 0,Y 500.037,Z 707.603,A -85,B 0,C 180,E1 -4791.835,E2 -4791.835} C_VEL
LIN {X 0,Y 501.074,Z 691.666,A -85,B 0,C 180,E1 -4793.397,E2 -4793.397} C_VEL
LIN {X 0,Y 502.192,Z 674.015,A -85,B 0,C 180,E1 -4794.842,E2 -4794.842} C_VEL
LIN {X 0,Y 503.256,Z 655.481,A -85,B 0,C 180,E1 -4796.101,E2 -4796.101} C_VEL
LIN {X 0,Y 504.197,Z 636.876,A -85,B 0,C 180,E1 -4797.137,E2 -4797.137} C_VEL
LIN {X 0,Y 505.11,Z 616.417,A -85,B 0,C 180,E1 -4798.044,E2 -4798.044} C_VEL
LIN {X 0,Y 505.853,Z 595.464,A -85,B 0,C 180,E1 -4798.742,E2 -4798.742} C_VEL
LIN {X 0,Y 506.394,Z 574.481,A -85,B 0,C 180,E1 -4799.226,E2 -4799.226} C_VEL
LIN {X 0,Y 508.288,Z 392.914,A -85,B 0,C 180,E1 -4801.962,E2 -4801.962} C_VEL
LIN {X 0,Y 509.019,Z 331.819,A -85,B 0,C 180,E1 -4802.967,E2 -4802.967} C_VEL
LIN {X 0,Y 506.9,Z 317.552,A -85,B 0,C 180,E1 -4803.39,E2 -4803.39} C_VEL
LIN {X 0,Y 507.597,Z 303.416,A -85,B 0,C 180,E1 -4804.477,E2 -4804.477} C_VEL
LIN {X 0,Y 501.679,Z 286.882,A -85,B 0,C 180,E1 -4806.437,E2 -4806.437} C_VEL
LIN {X 0,Y 498.35,Z 278.58,A -85,B 0,C 180,E1 -4807.585,E2 -4807.585} C_VEL
LIN {X 0,Y 496.787,Z 274.85,A -85,B 0,C 180,E1 -4808.204,E2 -4808.204} C_VEL
LIN {X 0,Y 496.734,Z 274.612,A -85,B 0,C 180,E1 -4811.689,E2 -4811.689} C_VEL
LIN {X 0,Y 496.754,Z 274.611,A -85,B 0,C 180,E1 -4815.213,E2 -4815.213} C_VEL
LIN {X 0,Y 496.775,Z 274.607,A -85,B 0,C 180,E1 -4818.688,E2 -4818.688} C_VEL
LIN {X 0,Y 496.735,Z 274.612,A -85,B 0,C 180,E1 -4822.127,E2 -4822.127} C_VEL
LIN {X 0,Y 496.768,Z 274.901,A -85,B 0,C 180,E1 -4823.9,E2 -4823.9} C_VEL
LIN {X 0,Y 500.068,Z 282.968,A -85,B 0,C 180,E1 -4825.264,E2 -4825.264} C_VEL
LIN {X 0,Y 504.417,Z 294.778,A -85,B 0,C 180,E1 -4826.968,E2 -4826.968} C_VEL
LIN {X 0,Y 506.659,Z 302.39,A -85,B 0,C 180,E1 -4827.937,E2 -4827.937} C_VEL
LIN {X 0,Y 504.302,Z 341.082,A -85,B 0,C 180,E1 -4831.423,E2 -4831.423} C_VEL
LIN {X 0,Y 507.189,Z 359.883,A -85,B 0,C 180,E1 -4831.992,E2 -4831.992} C_VEL
LIN {X 0,Y 505.208,Z 474.152,A -85,B 0,C 180,E1 -4833.848,E2 -4833.848} C_VEL
LIN {X 0,Y 504.179,Z 561.011,A -85,B 0,C 180,E1 -4835.197,E2 -4835.197} C_VEL
LIN {X 0,Y 503.6,Z 581.084,A -85,B 0,C 180,E1 -4835.727,E2 -4835.727} C_VEL
LIN {X 0,Y 502.863,Z 599.834,A -85,B 0,C 180,E1 -4836.444,E2 -4836.444} C_VEL
LIN {X 0,Y 501.968,Z 618.446,A -85,B 0,C 180,E1 -4837.392,E2 -4837.392} C_VEL
LIN {X 0,Y 501.011,Z 635.928,A -85,B 0,C 180,E1 -4838.518,E2 -4838.518} C_VEL
LIN {X 0,Y 500.015,Z 652.165,A -85,B 0,C 180,E1 -4839.822,E2 -4839.822} C_VEL
LIN {X 0,Y 498.991,Z 668.376,A -85,B 0,C 180,E1 -4841.404,E2 -4841.404} C_VEL
LIN {X 0,Y 498.163,Z 681.6,A -85,B 0,C 180,E1 -4842.961,E2 -4842.961} C_VEL
LIN {X 0,Y 497.426,Z 694.289,A -85,B 0,C 180,E1 -4844.733,E2 -4844.733} C_VEL
LIN {X 0,Y 496.85,Z 705.515,A -85,B 0,C 180,E1 -4846.619,E2 -4846.619} C_VEL
LIN {X 0,Y 496.427,Z 715.203,A -85,B 0,C 180,E1 -4848.616,E2 -4848.616} C_VEL
LIN {X 0,Y 496.162,Z 722.983,A -85,B 0,C 180,E1 -4850.606,E2 -4850.606} C_VEL
LIN {X 0,Y 496.006,Z 729.436,A -85,B 0,C 180,E1 -4852.704,E2 -4852.704} C_VEL
LIN {X 0,Y 495.94,Z 734.373,A -85,B 0,C 180,E1 -4854.911,E2 -4854.911} C_VEL
LIN {X 0,Y 495.914,Z 737.458,A -85,B 0,C 180,E1 -4857.111,E2 -4857.111} C_VEL
LIN {X 0,Y 495.914,Z 738.85,A -85,B 0,C 180,E1 -4859.307,E2 -4859.307} C_VEL
LIN {X 0,Y 495.91,Z 738.609,A -85,B 0,C 180,E1 -4861.502,E2 -4861.502} C_VEL
LIN {X 0,Y 495.912,Z 736.657,A -85,B 0,C 180,E1 -4863.7,E2 -4863.7} C_VEL
LIN {X 0,Y 495.949,Z 732.923,A -85,B 0,C 180,E1 -4865.902,E2 -4865.902} C_VEL
LIN {X 0,Y 496.049,Z 727.391,A -85,B 0,C 180,E1 -4868.112,E2 -4868.112} C_VEL
LIN {X 0,Y 496.238,Z 720.359,A -85,B 0,C 180,E1 -4870.214,E2 -4870.214} C_VEL
LIN {X 0,Y 496.56,Z 711.892,A -85,B 0,C 180,E1 -4872.206,E2 -4872.206} C_VEL
LIN {X 0,Y 497.034,Z 701.633,A -85,B 0,C 180,E1 -4874.158,E2 -4874.158} C_VEL
LIN {X 0,Y 497.658,Z 690.096,A -85,B 0,C 180,E1 -4875.977,E2 -4875.977} C_VEL
LIN {X 0,Y 498.427,Z 677.376,A -85,B 0,C 180,E1 -4877.66,E2 -4877.66} C_VEL
LIN {X 0,Y 499.319,Z 663.137,A -85,B 0,C 180,E1 -4879.233,E2 -4879.233} C_VEL
LIN {X 0,Y 500.335,Z 646.924,A -85,B 0,C 180,E1 -4880.715,E2 -4880.715} C_VEL
LIN {X 0,Y 501.337,Z 630.264,A -85,B 0,C 180,E1 -4881.967,E2 -4881.967} C_VEL
LIN {X 0,Y 502.287,Z 612.613,A -85,B 0,C 180,E1 -4883.027,E2 -4883.027} C_VEL
LIN {X 0,Y 503.176,Z 593.403,A -85,B 0,C 180,E1 -4883.926,E2 -4883.926} C_VEL
LIN {X 0,Y 503.874,Z 574.138,A -85,B 0,C 180,E1 -4884.589,E2 -4884.589} C_VEL
LIN {X 0,Y 504.363,Z 554.443,A -85,B 0,C 180,E1 -4885.034,E2 -4885.034} C_VEL
LIN {X 0,Y 506.641,Z 358.228,A -85,B 0,C 180,E1 -4888.032,E2 -4888.032} C_VEL
LIN {X 0,Y 505.059,Z 353.42,A -85,B 0,C 180,E1 -4888.219,E2 -4888.219} C_VEL
LIN {X 0,Y 499.919,Z 345.851,A -85,B 0,C 180,E1 -4888.685,E2 -4888.685} C_VEL
LIN {X 0,Y 497.214,Z 341.288,A -85,B 0,C 180,E1 -4889.015,E2 -4889.015} C_VEL
LIN {X 0,Y 496.832,Z 338.92,A -85,B 0,C 180,E1 -4889.213,E2 -4889.213} C_VEL
LIN {X 0,Y 498.75,Z 303.753,A -85,B 0,C 180,E1 -4892.362,E2 -4892.362} C_VEL
LIN {X 0,Y 491.879,Z 284.216,A -85,B 0,C 180,E1 -4894.791,E2 -4894.791} C_VEL
LIN {X 0,Y 488.822,Z 275.791,A -85,B 0,C 180,E1 -4895.941,E2 -4895.941} C_VEL
LIN {X 0,Y 488.834,Z 275.59,A -85,B 0,C 180,E1 -4899.36,E2 -4899.36} C_VEL
LIN {X 0,Y 488.83,Z 275.597,A -85,B 0,C 180,E1 -4902.932,E2 -4902.932} C_VEL
LIN {X 0,Y 488.823,Z 275.593,A -85,B 0,C 180,E1 -4906.564,E2 -4906.564} C_VEL
LIN {X 0,Y 488.818,Z 275.596,A -85,B 0,C 180,E1 -4910.09,E2 -4910.09} C_VEL
LIN {X 0,Y 488.828,Z 275.591,A -85,B 0,C 180,E1 -4913.698,E2 -4913.698} C_VEL
LIN {X 0,Y 488.814,Z 275.593,A -85,B 0,C 180,E1 -4917.214,E2 -4917.214} C_VEL
LIN {X 0,Y 488.806,Z 275.588,A -85,B 0,C 180,E1 -4920.866,E2 -4920.866} C_VEL
LIN {X 0,Y 488.82,Z 275.588,A -85,B 0,C 180,E1 -4924.43,E2 -4924.43} C_VEL
LIN {X 0,Y 488.836,Z 275.591,A -85,B 0,C 180,E1 -4928.018,E2 -4928.018} C_VEL
LIN {X 0,Y 488.804,Z 275.594,A -85,B 0,C 180,E1 -4931.514,E2 -4931.514} C_VEL
LIN {X 0,Y 488.771,Z 275.58,A -85,B 0,C 180,E1 -4934.941,E2 -4934.941} C_VEL
LIN {X 0,Y 488.803,Z 275.676,A -85,B 0,C 180,E1 -4938.315,E2 -4938.315} C_VEL
LIN {X 0,Y 489.195,Z 277.342,A -85,B 0,C 180,E1 -4938.564,E2 -4938.564} C_VEL
LIN {X 0,Y 495.993,Z 297.471,A -85,B 0,C 180,E1 -4940.718,E2 -4940.718} C_VEL
LIN {X 0,Y 496.654,Z 300.627,A -85,B 0,C 180,E1 -4941.023,E2 -4941.023} C_VEL
LIN {X 0,Y 495.796,Z 341.958,A -85,B 0,C 180,E1 -4944.444,E2 -4944.444} C_VEL
LIN {X 0,Y 494.775,Z 382.728,A -85,B 0,C 180,E1 -4947.798,E2 -4947.798} C_VEL
LIN {X 0,Y 493.521,Z 426.283,A -85,B 0,C 180,E1 -4951.392,E2 -4951.392} C_VEL
LIN {X 0,Y 492.405,Z 467.332,A -85,B 0,C 180,E1 -4954.774,E2 -4954.774} C_VEL
LIN {X 0,Y 492.302,Z 475.276,A -85,B 0,C 180,E1 -4955.378,E2 -4955.378} C_VEL
LIN {X 0,Y 493.414,Z 486.66,A -85,B 0,C 180,E1 -4955.599,E2 -4955.599} C_VEL
LIN {X 0,Y 492.302,Z 617.759,A -85,B 0,C 180,E1 -4957.57,E2 -4957.57} C_VEL
LIN {X 0,Y 491.997,Z 633.675,A -85,B 0,C 180,E1 -4958.023,E2 -4958.023} C_VEL
LIN {X 0,Y 491.529,Z 649.708,A -85,B 0,C 180,E1 -4958.709,E2 -4958.709} C_VEL
LIN {X 0,Y 490.98,Z 664.147,A -85,B 0,C 180,E1 -4959.552,E2 -4959.552} C_VEL
LIN {X 0,Y 490.347,Z 678.333,A -85,B 0,C 180,E1 -4960.627,E2 -4960.627} C_VEL
LIN {X 0,Y 489.798,Z 690.444,A -85,B 0,C 180,E1 -4961.778,E2 -4961.778} C_VEL
LIN {X 0,Y 489.211,Z 702.633,A -85,B 0,C 180,E1 -4963.231,E2 -4963.231} C_VEL
LIN {X 0,Y 488.771,Z 712.504,A -85,B 0,C 180,E1 -4964.693,E2 -4964.693} C_VEL
LIN {X 0,Y 488.399,Z 721.62,A -85,B 0,C 180,E1 -4966.409,E2 -4966.409} C_VEL
LIN {X 0,Y 488.172,Z 728.757,A -85,B 0,C 180,E1 -4968.137,E2 -4968.137} C_VEL
LIN {X 0,Y 488.035,Z 734.364,A -85,B 0,C 180,E1 -4970.006,E2 -4970.006} C_VEL
LIN {X 0,Y 487.976,Z 738.186,A -85,B 0,C 180,E1 -4971.894,E2 -4971.894} C_VEL
LIN {X 0,Y 487.956,Z 740.184,A -85,B 0,C 180,E1 -4973.806,E2 -4973.806} C_VEL
LIN {X 0,Y 487.954,Z 740.463,A -85,B 0,C 180,E1 -4975.746,E2 -4975.746} C_VEL
LIN {X 0,Y 487.967,Z 739.029,A -85,B 0,C 180,E1 -4977.584,E2 -4977.584} C_VEL
LIN {X 0,Y 488.015,Z 735.602,A -85,B 0,C 180,E1 -4979.587,E2 -4979.587} C_VEL
LIN {X 0,Y 488.119,Z 730.832,A -85,B 0,C 180,E1 -4981.35,E2 -4981.35} C_VEL
LIN {X 0,Y 488.321,Z 724.137,A -85,B 0,C 180,E1 -4983.139,E2 -4983.139} C_VEL
LIN {X 0,Y 488.636,Z 715.973,A -85,B 0,C 180,E1 -4984.811,E2 -4984.811} C_VEL
LIN {X 0,Y 489.088,Z 705.62,A -85,B 0,C 180,E1 -4986.463,E2 -4986.463} C_VEL
LIN {X 0,Y 489.608,Z 694.729,A -85,B 0,C 180,E1 -4987.853,E2 -4987.853} C_VEL
LIN {X 0,Y 490.22,Z 681.581,A -85,B 0,C 180,E1 -4989.189,E2 -4989.189} C_VEL
LIN {X 0,Y 490.835,Z 668.041,A -85,B 0,C 180,E1 -4990.28,E2 -4990.28} C_VEL
LIN {X 0,Y 491.443,Z 652.629,A -85,B 0,C 180,E1 -4991.236,E2 -4991.236} C_VEL
LIN {X 0,Y 491.923,Z 637.265,A -85,B 0,C 180,E1 -4991.939,E2 -4991.939} C_VEL
LIN {X 0,Y 492.26,Z 620.466,A -85,B 0,C 180,E1 -4992.462,E2 -4992.462} C_VEL
LIN {X 0,Y 492.473,Z 597.604,A -85,B 0,C 180,E1 -4992.851,E2 -4992.851} C_VEL
LIN {X 0,Y 493.242,Z 483.022,A -85,B 0,C 180,E1 -4994.558,E2 -4994.558} C_VEL
LIN {X 0,Y 492.238,Z 474.376,A -85,B 0,C 180,E1 -4994.771,E2 -4994.771} C_VEL
LIN {X 0,Y 493.397,Z 430.05,A -85,B 0,C 180,E1 -4998.395,E2 -4998.395} C_VEL
LIN {X 0,Y 494.609,Z 387.909,A -85,B 0,C 180,E1 -5001.844,E2 -5001.844} C_VEL
LIN {X 0,Y 495.441,Z 344.839,A -85,B 0,C 180,E1 -5005.311,E2 -5005.311} C_VEL
LIN {X 0,Y 496.02,Z 306.668,A -85,B 0,C 180,E1 -5008.392,E2 -5008.392} C_VEL
LIN {X 0,Y 495.9,Z 297.676,A -85,B 0,C 180,E1 -5009.126,E2 -5009.126} C_VEL
LIN {X 0,Y 489.365,Z 277.73,A -85,B 0,C 180,E1 -5011.171,E2 -5011.171} C_VEL
LIN {X 0,Y 488.811,Z 275.772,A -85,B 0,C 180,E1 -5011.433,E2 -5011.433} C_VEL
LIN {X 0,Y 488.819,Z 275.596,A -85,B 0,C 180,E1 -5014.82,E2 -5014.82} C_VEL
LIN {X 0,Y 488.834,Z 275.592,A -85,B 0,C 180,E1 -5018.397,E2 -5018.397} C_VEL
LIN {X 0,Y 488.797,Z 275.593,A -85,B 0,C 180,E1 -5021.885,E2 -5021.885} C_VEL
LIN {X 0,Y 488.79,Z 275.595,A -85,B 0,C 180,E1 -5025.427,E2 -5025.427} C_VEL
LIN {X 0,Y 488.823,Z 275.593,A -85,B 0,C 180,E1 -5028.914,E2 -5028.914} C_VEL
LIN {X 0,Y 488.834,Z 275.597,A -85,B 0,C 180,E1 -5032.478,E2 -5032.478} C_VEL
LIN {X 0,Y 488.799,Z 275.597,A -85,B 0,C 180,E1 -5036.012,E2 -5036.012} C_VEL
LIN {X 0,Y 488.793,Z 275.596,A -85,B 0,C 180,E1 -5039.648,E2 -5039.648} C_VEL
LIN {X 0,Y 488.817,Z 275.592,A -85,B 0,C 180,E1 -5043.166,E2 -5043.166} C_VEL
LIN {X 0,Y 488.833,Z 275.593,A -85,B 0,C 180,E1 -5046.695,E2 -5046.695} C_VEL
LIN {X 0,Y 488.806,Z 275.594,A -85,B 0,C 180,E1 -5050.251,E2 -5050.251} C_VEL
LIN {X 0,Y 488.794,Z 275.595,A -85,B 0,C 180,E1 -5053.847,E2 -5053.847} C_VEL
LIN {X 0,Y 488.816,Z 275.593,A -85,B 0,C 180,E1 -5057.375,E2 -5057.375} C_VEL
LIN {X 0,Y 488.835,Z 275.592,A -85,B 0,C 180,E1 -5060.974,E2 -5060.974} C_VEL
LIN {X 0,Y 488.819,Z 275.597,A -85,B 0,C 180,E1 -5064.533,E2 -5064.533} C_VEL
LIN {X 0,Y 488.797,Z 275.595,A -85,B 0,C 180,E1 -5068.065,E2 -5068.065} C_VEL
LIN {X 0,Y 488.814,Z 275.592,A -85,B 0,C 180,E1 -5071.577,E2 -5071.577} C_VEL
LIN {X 0,Y 488.833,Z 275.594,A -85,B 0,C 180,E1 -5075.102,E2 -5075.102} C_VEL
LIN {X 0,Y 488.828,Z 275.598,A -85,B 0,C 180,E1 -5078.748,E2 -5078.748} C_VEL
LIN {X 0,Y 488.802,Z 275.598,A -85,B 0,C 180,E1 -5082.297,E2 -5082.297} C_VEL
LIN {X 0,Y 488.806,Z 275.595,A -85,B 0,C 180,E1 -5085.937,E2 -5085.937} C_VEL
LIN {X 0,Y 488.832,Z 275.595,A -85,B 0,C 180,E1 -5089.542,E2 -5089.542} C_VEL
LIN {X 0,Y 488.869,Z 275.852,A -85,B 0,C 180,E1 -5091.446,E2 -5091.446} C_VEL
LIN {X 0,Y 492.109,Z 284.143,A -85,B 0,C 180,E1 -5092.505,E2 -5092.505} C_VEL
LIN {X 0,Y 500.017,Z 304.476,A -85,B 0,C 180,E1 -5094.87,E2 -5094.87} C_VEL
LIN {X 0,Y 500.977,Z 307.529,A -85,B 0,C 180,E1 -5095.196,E2 -5095.196} C_VEL
LIN {X 0,Y 500.587,Z 316.917,A -85,B 0,C 180,E1 -5095.891,E2 -5095.891} C_VEL
LIN {X 0,Y 503.315,Z 335.797,A -85,B 0,C 180,E1 -5096.438,E2 -5096.438} C_VEL
LIN {X 0,Y 501.332,Z 459.092,A -85,B 0,C 180,E1 -5098.416,E2 -5098.416} C_VEL
LIN {X 0,Y 499.699,Z 577.734,A -85,B 0,C 180,E1 -5100.285,E2 -5100.285} C_VEL
LIN {X 0,Y 498.941,Z 599.291,A -85,B 0,C 180,E1 -5100.841,E2 -5100.841} C_VEL
LIN {X 0,Y 498.031,Z 619.627,A -85,B 0,C 180,E1 -5101.59,E2 -5101.59} C_VEL
LIN {X 0,Y 496.93,Z 639.428,A -85,B 0,C 180,E1 -5102.538,E2 -5102.538} C_VEL
LIN {X 0,Y 495.733,Z 658.737,A -85,B 0,C 180,E1 -5103.697,E2 -5103.697} C_VEL
LIN {X 0,Y 494.467,Z 677.403,A -85,B 0,C 180,E1 -5105.064,E2 -5105.064} C_VEL
LIN {X 0,Y 493.206,Z 694.771,A -85,B 0,C 180,E1 -5106.59,E2 -5106.59} C_VEL
LIN {X 0,Y 492.068,Z 710.441,A -85,B 0,C 180,E1 -5108.217,E2 -5108.217} C_VEL
LIN {X 0,Y 491.027,Z 725.018,A -85,B 0,C 180,E1 -5109.997,E2 -5109.997} C_VEL
LIN {X 0,Y 490.151,Z 737.581,A -85,B 0,C 180,E1 -5111.816,E2 -5111.816} C_VEL
LIN {X 0,Y 489.358,Z 749.381,A -85,B 0,C 180,E1 -5113.868,E2 -5113.868} C_VEL
LIN {X 0,Y 488.733,Z 760.337,A -85,B 0,C 180,E1 -5116.153,E2 -5116.153} C_VEL
LIN {X 0,Y 488.326,Z 769.254,A -85,B 0,C 180,E1 -5118.426,E2 -5118.426} C_VEL
LIN {X 0,Y 488.086,Z 776.378,A -85,B 0,C 180,E1 -5120.688,E2 -5120.688} C_VEL
LIN {X 0,Y 487.968,Z 782.008,A -85,B 0,C 180,E1 -5123.058,E2 -5123.058} C_VEL
LIN {X 0,Y 487.919,Z 785.928,A -85,B 0,C 180,E1 -5125.417,E2 -5125.417} C_VEL
LIN {X 0,Y 487.91,Z 788.305,A -85,B 0,C 180,E1 -5127.887,E2 -5127.887} C_VEL
LIN {X 0,Y 487.906,Z 788.962,A -85,B 0,C 180,E1 -5130.236,E2 -5130.236} C_VEL
LIN {X 0,Y 487.909,Z 788.03,A -85,B 0,C 180,E1 -5132.585,E2 -5132.585} C_VEL
LIN {X 0,Y 487.924,Z 785.444,A -85,B 0,C 180,E1 -5134.939,E2 -5134.939} C_VEL
LIN {X 0,Y 487.972,Z 781.241,A -85,B 0,C 180,E1 -5137.3,E2 -5137.3} C_VEL
LIN {X 0,Y 488.119,Z 775.322,A -85,B 0,C 180,E1 -5139.671,E2 -5139.671} C_VEL
LIN {X 0,Y 488.381,Z 768.004,A -85,B 0,C 180,E1 -5141.935,E2 -5141.935} C_VEL
LIN {X 0,Y 488.815,Z 758.782,A -85,B 0,C 180,E1 -5144.21,E2 -5144.21} C_VEL
LIN {X 0,Y 489.44,Z 748.097,A -85,B 0,C 180,E1 -5146.376,E2 -5146.376} C_VEL
LIN {X 0,Y 490.254,Z 736.008,A -85,B 0,C 180,E1 -5148.429,E2 -5148.429} C_VEL
LIN {X 0,Y 491.139,Z 722.949,A -85,B 0,C 180,E1 -5150.249,E2 -5150.249} C_VEL
LIN {X 0,Y 492.149,Z 708.555,A -85,B 0,C 180,E1 -5151.952,E2 -5151.952} C_VEL
LIN {X 0,Y 493.292,Z 691.729,A -85,B 0,C 180,E1 -5153.629,E2 -5153.629} C_VEL
LIN {X 0,Y 494.425,Z 674.742,A -85,B 0,C 180,E1 -5155.046,E2 -5155.046} C_VEL
LIN {X 0,Y 495.528,Z 656.63,A -85,B 0,C 180,E1 -5156.308,E2 -5156.308} C_VEL
LIN {X 0,Y 496.623,Z 636.444,A -85,B 0,C 180,E1 -5157.456,E2 -5157.456} C_VEL
LIN {X 0,Y 497.584,Z 615.889,A -85,B 0,C 180,E1 -5158.375,E2 -5158.375} C_VEL
LIN {X 0,Y 498.379,Z 594.842,A -85,B 0,C 180,E1 -5159.081,E2 -5159.081} C_VEL
LIN {X 0,Y 498.936,Z 573.868,A -85,B 0,C 180,E1 -5159.567,E2 -5159.567} C_VEL
LIN {X 0,Y 500.822,Z 412.071,A -85,B 0,C 180,E1 -5162.054,E2 -5162.054} C_VEL
LIN {X 0,Y 502.027,Z 333.036,A -85,B 0,C 180,E1 -5163.397,E2 -5163.397} C_VEL
LIN {X 0,Y 499.908,Z 318.175,A -85,B 0,C 180,E1 -5163.858,E2 -5163.858} C_VEL
LIN {X 0,Y 500.482,Z 306.301,A -85,B 0,C 180,E1 -5164.806,E2 -5164.806} C_VEL
LIN {X 0,Y 495.135,Z 290.88,A -85,B 0,C 180,E1 -5166.709,E2 -5166.709} C_VEL
LIN {X 0,Y 491.749,Z 282.725,A -85,B 0,C 180,E1 -5167.917,E2 -5167.917} C_VEL
LIN {X 0,Y 489.923,Z 278.74,A -85,B 0,C 180,E1 -5168.589,E2 -5168.589} C_VEL
LIN {X 0,Y 488.841,Z 275.757,A -85,B 0,C 180,E1 -5169.178,E2 -5169.178} C_VEL
LIN {X 0,Y 488.834,Z 275.597,A -85,B 0,C 180,E1 -5172.753,E2 -5172.753} C_VEL
LIN {X 0,Y 488.81,Z 275.599,A -85,B 0,C 180,E1 -5176.261,E2 -5176.261} C_VEL
LIN {X 0,Y 488.79,Z 275.601,A -85,B 0,C 180,E1 -5179.731,E2 -5179.731} C_VEL
LIN {X 0,Y 488.863,Z 275.824,A -85,B 0,C 180,E1 -5182.908,E2 -5182.908} C_VEL
LIN {X 0,Y 490.357,Z 279.478,A -85,B 0,C 180,E1 -5183.652,E2 -5183.652} C_VEL
LIN {X 0,Y 493.795,Z 287.723,A -85,B 0,C 180,E1 -5185.092,E2 -5185.092} C_VEL
LIN {X 0,Y 497.768,Z 298.786,A -85,B 0,C 180,E1 -5186.745,E2 -5186.745} C_VEL
LIN {X 0,Y 499.736,Z 305.187,A -85,B 0,C 180,E1 -5187.601,E2 -5187.601} C_VEL
LIN {X 0,Y 497.286,Z 340.623,A -85,B 0,C 180,E1 -5190.868,E2 -5190.868} C_VEL
LIN {X 0,Y 500.347,Z 360.709,A -85,B 0,C 180,E1 -5191.529,E2 -5191.529} C_VEL
LIN {X 0,Y 497.85,Z 485.366,A -85,B 0,C 180,E1 -5193.627,E2 -5193.627} C_VEL
LIN {X 0,Y 496.774,Z 561.777,A -85,B 0,C 180,E1 -5194.858,E2 -5194.858} C_VEL
LIN {X 0,Y 496.153,Z 581.613,A -85,B 0,C 180,E1 -5195.397,E2 -5195.397} C_VEL
LIN {X 0,Y 495.386,Z 599.933,A -85,B 0,C 180,E1 -5196.109,E2 -5196.109} C_VEL
LIN {X 0,Y 494.481,Z 617.922,A -85,B 0,C 180,E1 -5197.03,E2 -5197.03} C_VEL
LIN {X 0,Y 493.46,Z 635.51,A -85,B 0,C 180,E1 -5198.167,E2 -5198.167} C_VEL
LIN {X 0,Y 492.401,Z 652.08,A -85,B 0,C 180,E1 -5199.496,E2 -5199.496} C_VEL
LIN {X 0,Y 491.319,Z 667.984,A -85,B 0,C 180,E1 -5201.06,E2 -5201.06} C_VEL
LIN {X 0,Y 490.392,Z 681.604,A -85,B 0,C 180,E1 -5202.682,E2 -5202.682} C_VEL
LIN {X 0,Y 489.587,Z 694.29,A -85,B 0,C 180,E1 -5204.483,E2 -5204.483} C_VEL
LIN {X 0,Y 488.956,Z 705.523,A -85,B 0,C 180,E1 -5206.399,E2 -5206.399} C_VEL
LIN {X 0,Y 488.485,Z 715.203,A -85,B 0,C 180,E1 -5208.429,E2 -5208.429} C_VEL
LIN {X 0,Y 488.193,Z 722.984,A -85,B 0,C 180,E1 -5210.451,E2 -5210.451} C_VEL
LIN {X 0,Y 488.016,Z 729.439,A -85,B 0,C 180,E1 -5212.586,E2 -5212.586} C_VEL
LIN {X 0,Y 487.942,Z 734.377,A -85,B 0,C 180,E1 -5214.827,E2 -5214.827} C_VEL
LIN {X 0,Y 487.914,Z 737.456,A -85,B 0,C 180,E1 -5217.064,E2 -5217.064} C_VEL
LIN {X 0,Y 487.915,Z 738.848,A -85,B 0,C 180,E1 -5219.296,E2 -5219.296} C_VEL
LIN {X 0,Y 487.91,Z 738.609,A -85,B 0,C 180,E1 -5221.527,E2 -5221.527} C_VEL
LIN {X 0,Y 487.913,Z 736.653,A -85,B 0,C 180,E1 -5223.76,E2 -5223.76} C_VEL
LIN {X 0,Y 487.951,Z 733.154,A -85,B 0,C 180,E1 -5225.881,E2 -5225.881} C_VEL
LIN {X 0,Y 488.057,Z 727.733,A -85,B 0,C 180,E1 -5228.127,E2 -5228.127} C_VEL
LIN {X 0,Y 488.263,Z 720.817,A -85,B 0,C 180,E1 -5230.263,E2 -5230.263} C_VEL
LIN {X 0,Y 488.632,Z 711.886,A -85,B 0,C 180,E1 -5232.408,E2 -5232.408} C_VEL
LIN {X 0,Y 489.135,Z 702.017,A -85,B 0,C 180,E1 -5234.321,E2 -5234.321} C_VEL
LIN {X 0,Y 489.844,Z 690.087,A -85,B 0,C 180,E1 -5236.239,E2 -5236.239} C_VEL
LIN {X 0,Y 490.706,Z 677.104,A -85,B 0,C 180,E1 -5237.981,E2 -5237.981} C_VEL
LIN {X 0,Y 491.645,Z 663.277,A -85,B 0,C 180,E1 -5239.528,E2 -5239.528} C_VEL
LIN {X 0,Y 492.729,Z 647.16,A -85,B 0,C 180,E1 -5241.02,E2 -5241.02} C_VEL
LIN {X 0,Y 493.811,Z 630.211,A -85,B 0,C 180,E1 -5242.306,E2 -5242.306} C_VEL
LIN {X 0,Y 494.783,Z 613.369,A -85,B 0,C 180,E1 -5243.334,E2 -5243.334} C_VEL
LIN {X 0,Y 495.718,Z 594.597,A -85,B 0,C 180,E1 -5244.234,E2 -5244.234} C_VEL
LIN {X 0,Y 496.477,Z 575.311,A -85,B 0,C 180,E1 -5244.92,E2 -5244.92} C_VEL
LIN {X 0,Y 497.033,Z 555.361,A -85,B 0,C 180,E1 -5245.392,E2 -5245.392} C_VEL
LIN {X 0,Y 499.659,Z 359.486,A -85,B 0,C 180,E1 -5248.46,E2 -5248.46} C_VEL
LIN {X 0,Y 496.729,Z 341.654,A -85,B 0,C 180,E1 -5248.987,E2 -5248.987} C_VEL
LIN {X 0,Y 496.832,Z 338.92,A -85,B 0,C 180,E1 -5249.213,E2 -5249.213} C_VEL
LIN {X 0,Y 496.258,Z 333.047,A -85,B 0,C 180,E1 -5249.795,E2 -5249.795} C_VEL
LIN {X 0,Y 491.542,Z 318.436,A -85,B 0,C 180,E1 -5251.502,E2 -5251.502} C_VEL
LIN {X 0,Y 491.19,Z 313.389,A -85,B 0,C 180,E1 -5252.01,E2 -5252.01} C_VEL
LIN {X 0,Y 491.549,Z 306.605,A -85,B 0,C 180,E1 -5252.635,E2 -5252.635} C_VEL
LIN {X 0,Y 484.858,Z 287.583,A -85,B 0,C 180,E1 -5255.046,E2 -5255.046} C_VEL
LIN {X 0,Y 480.892,Z 276.792,A -85,B 0,C 180,E1 -5256.539,E2 -5256.539} C_VEL
LIN {X 0,Y 480.861,Z 276.584,A -85,B 0,C 180,E1 -5260.135,E2 -5260.135} C_VEL
LIN {X 0,Y 480.883,Z 276.581,A -85,B 0,C 180,E1 -5263.655,E2 -5263.655} C_VEL
LIN {X 0,Y 480.889,Z 276.582,A -85,B 0,C 180,E1 -5267.22,E2 -5267.22} C_VEL
LIN {X 0,Y 480.885,Z 276.586,A -85,B 0,C 180,E1 -5270.855,E2 -5270.855} C_VEL
LIN {X 0,Y 480.887,Z 276.586,A -85,B 0,C 180,E1 -5274.395,E2 -5274.395} C_VEL
LIN {X 0,Y 480.89,Z 276.583,A -85,B 0,C 180,E1 -5278.029,E2 -5278.029} C_VEL
LIN {X 0,Y 480.888,Z 276.575,A -85,B 0,C 180,E1 -5281.583,E2 -5281.583} C_VEL
LIN {X 0,Y 480.859,Z 276.576,A -85,B 0,C 180,E1 -5285.163,E2 -5285.163} C_VEL
LIN {X 0,Y 480.852,Z 276.58,A -85,B 0,C 180,E1 -5288.788,E2 -5288.788} C_VEL
LIN {X 0,Y 480.869,Z 276.581,A -85,B 0,C 180,E1 -5292.327,E2 -5292.327} C_VEL
LIN {X 0,Y 480.891,Z 276.549,A -85,B 0,C 180,E1 -5295.92,E2 -5295.92} C_VEL
LIN {X 0,Y 480.918,Z 276.848,A -85,B 0,C 180,E1 -5297.906,E2 -5297.906} C_VEL
LIN {X 0,Y 488.444,Z 299.45,A -85,B 0,C 180,E1 -5300.395,E2 -5300.395} C_VEL
LIN {X 0,Y 489.329,Z 303.139,A -85,B 0,C 180,E1 -5300.769,E2 -5300.769} C_VEL
LIN {X 0,Y 488.397,Z 344.101,A -85,B 0,C 180,E1 -5304.183,E2 -5304.183} C_VEL
LIN {X 0,Y 487.266,Z 385.057,A -85,B 0,C 180,E1 -5307.588,E2 -5307.588} C_VEL
LIN {X 0,Y 485.959,Z 428.308,A -85,B 0,C 180,E1 -5311.178,E2 -5311.178} C_VEL
LIN {X 0,Y 484.782,Z 468.905,A -85,B 0,C 180,E1 -5314.553,E2 -5314.553} C_VEL
LIN {X 0,Y 484.71,Z 475.67,A -85,B 0,C 180,E1 -5315.062,E2 -5315.062} C_VEL
LIN {X 0,Y 485.868,Z 487.443,A -85,B 0,C 180,E1 -5315.295,E2 -5315.295} C_VEL
LIN {X 0,Y 484.673,Z 618.138,A -85,B 0,C 180,E1 -5317.291,E2 -5317.291} C_VEL
LIN {X 0,Y 484.347,Z 634.096,A -85,B 0,C 180,E1 -5317.752,E2 -5317.752} C_VEL
LIN {X 0,Y 483.857,Z 649.838,A -85,B 0,C 180,E1 -5318.435,E2 -5318.435} C_VEL
LIN {X 0,Y 483.274,Z 664.307,A -85,B 0,C 180,E1 -5319.288,E2 -5319.288} C_VEL
LIN {X 0,Y 482.589,Z 678.583,A -85,B 0,C 180,E1 -5320.383,E2 -5320.383} C_VEL
LIN {X 0,Y 481.968,Z 691.229,A -85,B 0,C 180,E1 -5321.607,E2 -5321.607} C_VEL
LIN {X 0,Y 481.338,Z 703.356,A -85,B 0,C 180,E1 -5323.085,E2 -5323.085} C_VEL
LIN {X 0,Y 480.861,Z 713.157,A -85,B 0,C 180,E1 -5324.57,E2 -5324.57} C_VEL
LIN {X 0,Y 480.457,Z 722.223,A -85,B 0,C 180,E1 -5326.315,E2 -5326.315} C_VEL
LIN {X 0,Y 480.208,Z 729.304,A -85,B 0,C 180,E1 -5328.072,E2 -5328.072} C_VEL
LIN {X 0,Y 480.056,Z 734.869,A -85,B 0,C 180,E1 -5329.971,E2 -5329.971} C_VEL
LIN {X 0,Y 479.989,Z 738.645,A -85,B 0,C 180,E1 -5331.891,E2 -5331.891} C_VEL
LIN {X 0,Y 479.965,Z 740.614,A -85,B 0,C 180,E1 -5333.861,E2 -5333.861} C_VEL
LIN {X 0,Y 479.965,Z 740.831,A -85,B 0,C 180,E1 -5335.849,E2 -5335.849} C_VEL
LIN {X 0,Y 479.982,Z 739.18,A -85,B 0,C 180,E1 -5337.813,E2 -5337.813} C_VEL
LIN {X 0,Y 480.042,Z 735.885,A -85,B 0,C 180,E1 -5339.715,E2 -5339.715} C_VEL
LIN {X 0,Y 480.169,Z 730.727,A -85,B 0,C 180,E1 -5341.606,E2 -5341.606} C_VEL
LIN {X 0,Y 480.415,Z 723.707,A -85,B 0,C 180,E1 -5343.47,E2 -5343.47} C_VEL
LIN {X 0,Y 480.778,Z 715.173,A -85,B 0,C 180,E1 -5345.183,E2 -5345.183} C_VEL
LIN {X 0,Y 481.28,Z 704.964,A -85,B 0,C 180,E1 -5346.804,E2 -5346.804} C_VEL
LIN {X 0,Y 481.872,Z 693.376,A -85,B 0,C 180,E1 -5348.258,E2 -5348.258} C_VEL
LIN {X 0,Y 482.539,Z 680.323,A -85,B 0,C 180,E1 -5349.572,E2 -5349.572} C_VEL
LIN {X 0,Y 483.198,Z 666.3,A -85,B 0,C 180,E1 -5350.676,E2 -5350.676} C_VEL
LIN {X 0,Y 483.819,Z 651.659,A -85,B 0,C 180,E1 -5351.572,E2 -5351.572} C_VEL
LIN {X 0,Y 484.321,Z 635.548,A -85,B 0,C 180,E1 -5352.29,E2 -5352.29} C_VEL
LIN {X 0,Y 484.657,Z 619.372,A -85,B 0,C 180,E1 -5352.778,E2 -5352.778} C_VEL
LIN {X 0,Y 485.06,Z 573.604,A -85,B 0,C 180,E1 -5353.502,E2 -5353.502} C_VEL
LIN {X 0,Y 485.702,Z 483.779,A -85,B 0,C 180,E1 -5354.867,E2 -5354.867} C_VEL
LIN {X 0,Y 484.654,Z 474.864,A -85,B 0,C 180,E1 -5355.083,E2 -5355.083} C_VEL
LIN {X 0,Y 485.874,Z 430.646,A -85,B 0,C 180,E1 -5358.726,E2 -5358.726} C_VEL
LIN {X 0,Y 487.07,Z 390.003,A -85,B 0,C 180,E1 -5362.061,E2 -5362.061} C_VEL
LIN {X 0,Y 487.969,Z 349.682,A -85,B 0,C 180,E1 -5365.346,E2 -5365.346} C_VEL
LIN {X 0,Y 488.646,Z 311.158,A -85,B 0,C 180,E1 -5368.479,E2 -5368.479} C_VEL
LIN {X 0,Y 488.615,Z 300.388,A -85,B 0,C 180,E1 -5369.367,E2 -5369.367} C_VEL
LIN {X 0,Y 481.718,Z 279.355,A -85,B 0,C 180,E1 -5371.552,E2 -5371.552} C_VEL
LIN {X 0,Y 480.89,Z 276.79,A -85,B 0,C 180,E1 -5371.881,E2 -5371.881} C_VEL
LIN {X 0,Y 480.851,Z 276.59,A -85,B 0,C 180,E1 -5375.425,E2 -5375.425} C_VEL
LIN {X 0,Y 480.873,Z 276.581,A -85,B 0,C 180,E1 -5378.995,E2 -5378.995} C_VEL
LIN {X 0,Y 480.895,Z 276.586,A -85,B 0,C 180,E1 -5382.611,E2 -5382.611} C_VEL
LIN {X 0,Y 480.874,Z 276.588,A -85,B 0,C 180,E1 -5386.165,E2 -5386.165} C_VEL
LIN {X 0,Y 480.852,Z 276.585,A -85,B 0,C 180,E1 -5389.698,E2 -5389.698} C_VEL
LIN {X 0,Y 480.861,Z 276.582,A -85,B 0,C 180,E1 -5393.313,E2 -5393.313} C_VEL
LIN {X 0,Y 480.889,Z 276.583,A -85,B 0,C 180,E1 -5396.901,E2 -5396.901} C_VEL
LIN {X 0,Y 480.891,Z 276.584,A -85,B 0,C 180,E1 -5400.476,E2 -5400.476} C_VEL
LIN {X 0,Y 480.859,Z 276.584,A -85,B 0,C 180,E1 -5404.054,E2 -5404.054} C_VEL
LIN {X 0,Y 480.857,Z 276.583,A -85,B 0,C 180,E1 -5407.647,E2 -5407.647} C_VEL
LIN {X 0,Y 480.884,Z 276.582,A -85,B 0,C 180,E1 -5411.149,E2 -5411.149} C_VEL
LIN {X 0,Y 480.896,Z 276.581,A -85,B 0,C 180,E1 -5414.811,E2 -5414.811} C_VEL
LIN {X 0,Y 480.875,Z 276.586,A -85,B 0,C 180,E1 -5418.424,E2 -5418.424} C_VEL
LIN {X 0,Y 480.856,Z 276.582,A -85,B 0,C 180,E1 -5421.979,E2 -5421.979} C_VEL
LIN {X 0,Y 480.874,Z 276.582,A -85,B 0,C 180,E1 -5425.53,E2 -5425.53} C_VEL
LIN {X 0,Y 480.897,Z 276.579,A -85,B 0,C 180,E1 -5429.166,E2 -5429.166} C_VEL
LIN {X 0,Y 480.888,Z 276.586,A -85,B 0,C 180,E1 -5432.723,E2 -5432.723} C_VEL
LIN {X 0,Y 480.864,Z 276.585,A -85,B 0,C 180,E1 -5436.341,E2 -5436.341} C_VEL
LIN {X 0,Y 480.863,Z 276.584,A -85,B 0,C 180,E1 -5439.978,E2 -5439.978} C_VEL
LIN {X 0,Y 480.888,Z 276.584,A -85,B 0,C 180,E1 -5443.488,E2 -5443.488} C_VEL
LIN {X 0,Y 480.893,Z 276.584,A -85,B 0,C 180,E1 -5447.168,E2 -5447.168} C_VEL
LIN {X 0,Y 480.885,Z 276.658,A -85,B 0,C 180,E1 -5450.666,E2 -5450.666} C_VEL
LIN {X 0,Y 481.011,Z 277.282,A -85,B 0,C 180,E1 -5450.889,E2 -5450.889} C_VEL
LIN {X 0,Y 489.24,Z 297.693,A -85,B 0,C 180,E1 -5453.434,E2 -5453.434} C_VEL
LIN {X 0,Y 493.883,Z 310.615,A -85,B 0,C 180,E1 -5454.906,E2 -5454.906} C_VEL
LIN {X 0,Y 493.628,Z 317.053,A -85,B 0,C 180,E1 -5455.379,E2 -5455.379} C_VEL
LIN {X 0,Y 496.497,Z 336.987,A -85,B 0,C 180,E1 -5455.97,E2 -5455.97} C_VEL
LIN {X 0,Y 493.015,Z 543.06,A -85,B 0,C 180,E1 -5459.319,E2 -5459.319} C_VEL
LIN {X 0,Y 492.461,Z 578.367,A -85,B 0,C 180,E1 -5459.898,E2 -5459.898} C_VEL
LIN {X 0,Y 491.654,Z 599.684,A -85,B 0,C 180,E1 -5460.462,E2 -5460.462} C_VEL
LIN {X 0,Y 490.64,Z 620.714,A -85,B 0,C 180,E1 -5461.255,E2 -5461.255} C_VEL
LIN {X 0,Y 489.439,Z 640.672,A -85,B 0,C 180,E1 -5462.242,E2 -5462.242} C_VEL
LIN {X 0,Y 488.164,Z 659.689,A -85,B 0,C 180,E1 -5463.416,E2 -5463.416} C_VEL
LIN {X 0,Y 486.856,Z 677.606,A -85,B 0,C 180,E1 -5464.759,E2 -5464.759} C_VEL
LIN {X 0,Y 485.499,Z 695.057,A -85,B 0,C 180,E1 -5466.324,E2 -5466.324} C_VEL
LIN {X 0,Y 484.298,Z 710.567,A -85,B 0,C 180,E1 -5467.969,E2 -5467.969} C_VEL
LIN {X 0,Y 483.184,Z 725.151,A -85,B 0,C 180,E1 -5469.785,E2 -5469.785} C_VEL
LIN {X 0,Y 482.158,Z 739.298,A -85,B 0,C 180,E1 -5471.879,E2 -5471.879} C_VEL
LIN {X 0,Y 481.323,Z 751.868,A -85,B 0,C 180,E1 -5474.111,E2 -5474.111} C_VEL
LIN {X 0,Y 480.793,Z 760.85,A -85,B 0,C 180,E1 -5476.042,E2 -5476.042} C_VEL
LIN {X 0,Y 480.355,Z 769.658,A -85,B 0,C 180,E1 -5478.353,E2 -5478.353} C_VEL
LIN {X 0,Y 480.097,Z 776.687,A -85,B 0,C 180,E1 -5480.653,E2 -5480.653} C_VEL
LIN {X 0,Y 479.971,Z 782.262,A -85,B 0,C 180,E1 -5483.062,E2 -5483.062} C_VEL
LIN {X 0,Y 479.919,Z 786.088,A -85,B 0,C 180,E1 -5485.461,E2 -5485.461} C_VEL
LIN {X 0,Y 479.909,Z 788.304,A -85,B 0,C 180,E1 -5487.852,E2 -5487.852} C_VEL
LIN {X 0,Y 479.905,Z 788.961,A -85,B 0,C 180,E1 -5490.24,E2 -5490.24} C_VEL
LIN {X 0,Y 479.909,Z 788.029,A -85,B 0,C 180,E1 -5492.628,E2 -5492.628} C_VEL
LIN {X 0,Y 479.923,Z 785.444,A -85,B 0,C 180,E1 -5495.021,E2 -5495.021} C_VEL
LIN {X 0,Y 479.982,Z 781.182,A -85,B 0,C 180,E1 -5497.45,E2 -5497.45} C_VEL
LIN {X 0,Y 480.145,Z 775.322,A -85,B 0,C 180,E1 -5499.833,E2 -5499.833} C_VEL
LIN {X 0,Y 480.43,Z 768.003,A -85,B 0,C 180,E1 -5502.135,E2 -5502.135} C_VEL
LIN {X 0,Y 480.913,Z 758.779,A -85,B 0,C 180,E1 -5504.448,E2 -5504.448} C_VEL
LIN {X 0,Y 481.481,Z 749.052,A -85,B 0,C 180,E1 -5506.406,E2 -5506.406} C_VEL
LIN {X 0,Y 482.295,Z 736.669,A -85,B 0,C 180,E1 -5508.494,E2 -5508.494} C_VEL
LIN {X 0,Y 483.24,Z 723.261,A -85,B 0,C 180,E1 -5510.399,E2 -5510.399} C_VEL
LIN {X 0,Y 484.338,Z 708.311,A -85,B 0,C 180,E1 -5512.197,E2 -5512.197} C_VEL
LIN {X 0,Y 485.572,Z 691.104,A -85,B 0,C 180,E1 -5513.933,E2 -5513.933} C_VEL
LIN {X 0,Y 486.801,Z 673.363,A -85,B 0,C 180,E1 -5515.422,E2 -5515.422} C_VEL
LIN {X 0,Y 487.986,Z 654.951,A -85,B 0,C 180,E1 -5516.704,E2 -5516.704} C_VEL
LIN {X 0,Y 489.066,Z 636.002,A -85,B 0,C 180,E1 -5517.784,E2 -5517.784} C_VEL
LIN {X 0,Y 490.074,Z 615.351,A -85,B 0,C 180,E1 -5518.717,E2 -5518.717} C_VEL
LIN {X 0,Y 490.923,Z 594.202,A -85,B 0,C 180,E1 -5519.431,E2 -5519.431} C_VEL
LIN {X 0,Y 491.499,Z 573.212,A -85,B 0,C 180,E1 -5519.919,E2 -5519.919} C_VEL
LIN {X 0,Y 493.426,Z 427.106,A -85,B 0,C 180,E1 -5522.22,E2 -5522.22} C_VEL
LIN {X 0,Y 495.194,Z 334.57,A -85,B 0,C 180,E1 -5523.846,E2 -5523.846} C_VEL
LIN {X 0,Y 493.038,Z 318.591,A -85,B 0,C 180,E1 -5524.374,E2 -5524.374} C_VEL
LIN {X 0,Y 493.51,Z 309.486,A -85,B 0,C 180,E1 -5525.128,E2 -5525.128} C_VEL
LIN {X 0,Y 488.887,Z 295.609,A -85,B 0,C 180,E1 -5526.903,E2 -5526.903} C_VEL
LIN {X 0,Y 485.637,Z 287.551,A -85,B 0,C 180,E1 -5528.146,E2 -5528.146} C_VEL
LIN {X 0,Y 482.851,Z 280.995,A -85,B 0,C 180,E1 -5529.321,E2 -5529.321} C_VEL
LIN {X 0,Y 481.021,Z 277.436,A -85,B 0,C 180,E1 -5530.12,E2 -5530.12} C_VEL
LIN {X 0,Y 480.9,Z 276.647,A -85,B 0,C 180,E1 -5530.451,E2 -5530.451} C_VEL
LIN {X 0,Y 480.86,Z 276.588,A -85,B 0,C 180,E1 -5533.992,E2 -5533.992} C_VEL
LIN {X 0,Y 480.854,Z 276.59,A -85,B 0,C 180,E1 -5537.647,E2 -5537.647} C_VEL
LIN {X 0,Y 480.885,Z 276.587,A -85,B 0,C 180,E1 -5541.104,E2 -5541.104} C_VEL
LIN {X 0,Y 480.911,Z 276.996,A -85,B 0,C 180,E1 -5541.776,E2 -5541.776} C_VEL
LIN {X 0,Y 482.518,Z 280.522,A -85,B 0,C 180,E1 -5542.617,E2 -5542.617} C_VEL
LIN {X 0,Y 486.264,Z 289.034,A -85,B 0,C 180,E1 -5544.313,E2 -5544.313} C_VEL
LIN {X 0,Y 490.455,Z 300.635,A -85,B 0,C 180,E1 -5546.183,E2 -5546.183} C_VEL
LIN {X 0,Y 492.865,Z 308.324,A -85,B 0,C 180,E1 -5547.273,E2 -5547.273} C_VEL
LIN {X 0,Y 490.407,Z 340.423,A -85,B 0,C 180,E1 -5550.291,E2 -5550.291} C_VEL
LIN {X 0,Y 493.622,Z 361.673,A -85,B 0,C 180,E1 -5551.038,E2 -5551.038} C_VEL
LIN {X 0,Y 490.92,Z 469.402,A -85,B 0,C 180,E1 -5552.955,E2 -5552.955} C_VEL
LIN {X 0,Y 489.387,Z 562.174,A -85,B 0,C 180,E1 -5554.504,E2 -5554.504} C_VEL
LIN {X 0,Y 488.743,Z 581.455,A -85,B 0,C 180,E1 -5555.035,E2 -5555.035} C_VEL
LIN {X 0,Y 487.918,Z 600.195,A -85,B 0,C 180,E1 -5555.772,E2 -5555.772} C_VEL
LIN {X 0,Y 486.949,Z 618.418,A -85,B 0,C 180,E1 -5556.718,E2 -5556.718} C_VEL
LIN {X 0,Y 485.86,Z 636.052,A -85,B 0,C 180,E1 -5557.877,E2 -5557.877} C_VEL
LIN {X 0,Y 484.742,Z 652.559,A -85,B 0,C 180,E1 -5559.221,E2 -5559.221} C_VEL
LIN {X 0,Y 483.633,Z 667.932,A -85,B 0,C 180,E1 -5560.747,E2 -5560.747} C_VEL
LIN {X 0,Y 482.641,Z 681.672,A -85,B 0,C 180,E1 -5562.395,E2 -5562.395} C_VEL
LIN {X 0,Y 481.764,Z 694.357,A -85,B 0,C 180,E1 -5564.224,E2 -5564.224} C_VEL
LIN {X 0,Y 481.064,Z 705.528,A -85,B 0,C 180,E1 -5566.172,E2 -5566.172} C_VEL
LIN {X 0,Y 480.549,Z 715.203,A -85,B 0,C 180,E1 -5568.235,E2 -5568.235} C_VEL
LIN {X 0,Y 480.226,Z 722.986,A -85,B 0,C 180,E1 -5570.291,E2 -5570.291} C_VEL
LIN {X 0,Y 480.024,Z 729.574,A -85,B 0,C 180,E1 -5572.518,E2 -5572.518} C_VEL
LIN {X 0,Y 479.944,Z 734.41,A -85,B 0,C 180,E1 -5574.758,E2 -5574.758} C_VEL
LIN {X 0,Y 479.914,Z 737.453,A -85,B 0,C 180,E1 -5577.015,E2 -5577.015} C_VEL
LIN {X 0,Y 479.915,Z 738.847,A -85,B 0,C 180,E1 -5579.284,E2 -5579.284} C_VEL
LIN {X 0,Y 479.912,Z 738.677,A -85,B 0,C 180,E1 -5581.433,E2 -5581.433} C_VEL
LIN {X 0,Y 479.914,Z 736.777,A -85,B 0,C 180,E1 -5583.704,E2 -5583.704} C_VEL
LIN {X 0,Y 479.952,Z 733.384,A -85,B 0,C 180,E1 -5585.859,E2 -5585.859} C_VEL
LIN {X 0,Y 480.054,Z 728.422,A -85,B 0,C 180,E1 -5588.022,E2 -5588.022} C_VEL
LIN {X 0,Y 480.269,Z 721.665,A -85,B 0,C 180,E1 -5590.193,E2 -5590.193} C_VEL
LIN {X 0,Y 480.626,Z 713.468,A -85,B 0,C 180,E1 -5592.251,E2 -5592.251} C_VEL
LIN {X 0,Y 481.227,Z 702.728,A -85,B 0,C 180,E1 -5594.438,E2 -5594.438} C_VEL
LIN {X 0,Y 482.046,Z 690.126,A -85,B 0,C 180,E1 -5596.509,E2 -5596.509} C_VEL
LIN {X 0,Y 482.943,Z 677.594,A -85,B 0,C 180,E1 -5598.218,E2 -5598.218} C_VEL
LIN {X 0,Y 483.961,Z 663.643,A -85,B 0,C 180,E1 -5599.806,E2 -5599.806} C_VEL
LIN {X 0,Y 485.114,Z 647.635,A -85,B 0,C 180,E1 -5601.312,E2 -5601.312} C_VEL
LIN {X 0,Y 486.263,Z 630.749,A -85,B 0,C 180,E1 -5602.614,E2 -5602.614} C_VEL
LIN {X 0,Y 487.349,Z 612.991,A -85,B 0,C 180,E1 -5603.711,E2 -5603.711} C_VEL
LIN {X 0,Y 488.362,Z 594.03,A -85,B 0,C 180,E1 -5604.627,E2 -5604.627} C_VEL
LIN {X 0,Y 489.175,Z 574.432,A -85,B 0,C 180,E1 -5605.322,E2 -5605.322} C_VEL
LIN {X 0,Y 489.759,Z 554.493,A -85,B 0,C 180,E1 -5605.791,E2 -5605.791} C_VEL
LIN {X 0,Y 492.703,Z 360.753,A -85,B 0,C 180,E1 -5608.901,E2 -5608.901} C_VEL
LIN {X 0,Y 489.554,Z 341.423,A -85,B 0,C 180,E1 -5609.487,E2 -5609.487} C_VEL
LIN {X 0,Y 491.19,Z 313.389,A -85,B 0,C 180,E1 -5612.01,E2 -5612.01} C_VEL
LIN {X 0,Y 490.515,Z 310.28,A -85,B 0,C 180,E1 -5612.359,E2 -5612.359} C_VEL
LIN {X 0,Y 487.47,Z 306.792,A -85,B 0,C 180,E1 -5612.932,E2 -5612.932} C_VEL
LIN {X 0,Y 482.264,Z 302.171,A -85,B 0,C 180,E1 -5613.804,E2 -5613.804} C_VEL
LIN {X 0,Y 481.268,Z 300.303,A -85,B 0,C 180,E1 -5614.072,E2 -5614.072} C_VEL
LIN {X 0,Y 473.968,Z 280.663,A -85,B 0,C 180,E1 -5616.713,E2 -5616.713} C_VEL
LIN {X 0,Y 472.982,Z 277.764,A -85,B 0,C 180,E1 -5617.158,E2 -5617.158} C_VEL
LIN {X 0,Y 472.955,Z 277.574,A -85,B 0,C 180,E1 -5620.813,E2 -5620.813} C_VEL
LIN {X 0,Y 472.937,Z 277.569,A -85,B 0,C 180,E1 -5624.41,E2 -5624.41} C_VEL
LIN {X 0,Y 472.937,Z 277.574,A -85,B 0,C 180,E1 -5628.09,E2 -5628.09} C_VEL
LIN {X 0,Y 472.95,Z 277.57,A -85,B 0,C 180,E1 -5631.725,E2 -5631.725} C_VEL
LIN {X 0,Y 472.943,Z 277.57,A -85,B 0,C 180,E1 -5635.339,E2 -5635.339} C_VEL
LIN {X 0,Y 472.932,Z 277.57,A -85,B 0,C 180,E1 -5638.944,E2 -5638.944} C_VEL
LIN {X 0,Y 472.94,Z 277.577,A -85,B 0,C 180,E1 -5642.555,E2 -5642.555} C_VEL
LIN {X 0,Y 472.954,Z 277.568,A -85,B 0,C 180,E1 -5646.184,E2 -5646.184} C_VEL
LIN {X 0,Y 472.952,Z 277.57,A -85,B 0,C 180,E1 -5649.842,E2 -5649.842} C_VEL
LIN {X 0,Y 472.916,Z 277.578,A -85,B 0,C 180,E1 -5653.415,E2 -5653.415} C_VEL
LIN {X 0,Y 472.888,Z 277.551,A -85,B 0,C 180,E1 -5656.923,E2 -5656.923} C_VEL
LIN {X 0,Y 472.949,Z 277.865,A -85,B 0,C 180,E1 -5657.422,E2 -5657.422} C_VEL
LIN {X 0,Y 480.124,Z 299.048,A -85,B 0,C 180,E1 -5659.803,E2 -5659.803} C_VEL
LIN {X 0,Y 482.022,Z 305.695,A -85,B 0,C 180,E1 -5660.507,E2 -5660.507} C_VEL
LIN {X 0,Y 480.988,Z 346.959,A -85,B 0,C 180,E1 -5663.973,E2 -5663.973} C_VEL
LIN {X 0,Y 479.767,Z 388.214,A -85,B 0,C 180,E1 -5667.431,E2 -5667.431} C_VEL
LIN {X 0,Y 478.381,Z 431.042,A -85,B 0,C 180,E1 -5671.017,E2 -5671.017} C_VEL
LIN {X 0,Y 477.128,Z 471.961,A -85,B 0,C 180,E1 -5674.446,E2 -5674.446} C_VEL
LIN {X 0,Y 477.145,Z 476.184,A -85,B 0,C 180,E1 -5674.739,E2 -5674.739} C_VEL
LIN {X 0,Y 478.337,Z 488.23,A -85,B 0,C 180,E1 -5674.983,E2 -5674.983} C_VEL
LIN {X 0,Y 477.055,Z 618.508,A -85,B 0,C 180,E1 -5677.004,E2 -5677.004} C_VEL
LIN {X 0,Y 476.711,Z 634.427,A -85,B 0,C 180,E1 -5677.47,E2 -5677.47} C_VEL
LIN {X 0,Y 476.189,Z 650.185,A -85,B 0,C 180,E1 -5678.164,E2 -5678.164} C_VEL
LIN {X 0,Y 475.581,Z 664.381,A -85,B 0,C 180,E1 -5679.01,E2 -5679.01} C_VEL
LIN {X 0,Y 474.845,Z 678.749,A -85,B 0,C 180,E1 -5680.125,E2 -5680.125} C_VEL
LIN {X 0,Y 474.191,Z 691.16,A -85,B 0,C 180,E1 -5681.336,E2 -5681.336} C_VEL
LIN {X 0,Y 473.516,Z 703.151,A -85,B 0,C 180,E1 -5682.808,E2 -5682.808} C_VEL
LIN {X 0,Y 472.991,Z 713.077,A -85,B 0,C 180,E1 -5684.318,E2 -5684.318} C_VEL
LIN {X 0,Y 472.568,Z 721.663,A -85,B 0,C 180,E1 -5685.964,E2 -5685.964} C_VEL
LIN {X 0,Y 472.273,Z 728.948,A -85,B 0,C 180,E1 -5687.748,E2 -5687.748} C_VEL
LIN {X 0,Y 472.1,Z 734.434,A -85,B 0,C 180,E1 -5689.548,E2 -5689.548} C_VEL
LIN {X 0,Y 472.007,Z 738.604,A -85,B 0,C 180,E1 -5691.573,E2 -5691.573} C_VEL
LIN {X 0,Y 471.978,Z 740.795,A -85,B 0,C 180,E1 -5693.468,E2 -5693.468} C_VEL
LIN {X 0,Y 471.972,Z 741.29,A -85,B 0,C 180,E1 -5695.514,E2 -5695.514} C_VEL
LIN {X 0,Y 471.99,Z 740.026,A -85,B 0,C 180,E1 -5697.502,E2 -5697.502} C_VEL
LIN {X 0,Y 472.047,Z 736.922,A -85,B 0,C 180,E1 -5699.476,E2 -5699.476} C_VEL
LIN {X 0,Y 472.178,Z 732.074,A -85,B 0,C 180,E1 -5701.419,E2 -5701.419} C_VEL
LIN {X 0,Y 472.419,Z 725.464,A -85,B 0,C 180,E1 -5703.278,E2 -5703.278} C_VEL
LIN {X 0,Y 472.807,Z 717.11,A -85,B 0,C 180,E1 -5705.074,E2 -5705.074} C_VEL
LIN {X 0,Y 473.315,Z 707.291,A -85,B 0,C 180,E1 -5706.712,E2 -5706.712} C_VEL
LIN {X 0,Y 473.945,Z 696.083,A -85,B 0,C 180,E1 -5708.213,E2 -5708.213} C_VEL
LIN {X 0,Y 474.629,Z 683.459,A -85,B 0,C 180,E1 -5709.553,E2 -5709.553} C_VEL
LIN {X 0,Y 475.342,Z 670.013,A -85,B 0,C 180,E1 -5710.695,E2 -5710.695} C_VEL
LIN {X 0,Y 476.011,Z 655.204,A -85,B 0,C 180,E1 -5711.665,E2 -5711.665} C_VEL
LIN {X 0,Y 476.565,Z 640.458,A -85,B 0,C 180,E1 -5712.394,E2 -5712.394} C_VEL
LIN {X 0,Y 476.958,Z 624.513,A -85,B 0,C 180,E1 -5712.943,E2 -5712.943} C_VEL
LIN {X 0,Y 477.191,Z 606.756,A -85,B 0,C 180,E1 -5713.303,E2 -5713.303} C_VEL
LIN {X 0,Y 478.186,Z 484.616,A -85,B 0,C 180,E1 -5715.185,E2 -5715.185} C_VEL
LIN {X 0,Y 477.083,Z 475.353,A -85,B 0,C 180,E1 -5715.405,E2 -5715.405} C_VEL
LIN {X 0,Y 478.366,Z 431.489,A -85,B 0,C 180,E1 -5719.05,E2 -5719.05} C_VEL
LIN {X 0,Y 479.648,Z 390.654,A -85,B 0,C 180,E1 -5722.429,E2 -5722.429} C_VEL
LIN {X 0,Y 480.647,Z 348.534,A -85,B 0,C 180,E1 -5725.884,E2 -5725.884} C_VEL
LIN {X 0,Y 481.427,Z 308.035,A -85,B 0,C 180,E1 -5729.206,E2 -5729.206} C_VEL
LIN {X 0,Y 481.348,Z 303.12,A -85,B 0,C 180,E1 -5729.615,E2 -5729.615} C_VEL
LIN {X 0,Y 474.821,Z 283.199,A -85,B 0,C 180,E1 -5731.718,E2 -5731.718} C_VEL
LIN {X 0,Y 473,Z 277.889,A -85,B 0,C 180,E1 -5732.335,E2 -5732.335} C_VEL
LIN {X 0,Y 472.915,Z 277.578,A -85,B 0,C 180,E1 -5733.234,E2 -5733.234} C_VEL
LIN {X 0,Y 472.943,Z 277.572,A -85,B 0,C 180,E1 -5736.844,E2 -5736.844} C_VEL
LIN {X 0,Y 472.954,Z 277.571,A -85,B 0,C 180,E1 -5740.486,E2 -5740.486} C_VEL
LIN {X 0,Y 472.933,Z 277.572,A -85,B 0,C 180,E1 -5744.135,E2 -5744.135} C_VEL
LIN {X 0,Y 472.912,Z 277.575,A -85,B 0,C 180,E1 -5747.67,E2 -5747.67} C_VEL
LIN {X 0,Y 472.926,Z 277.571,A -85,B 0,C 180,E1 -5751.244,E2 -5751.244} C_VEL
LIN {X 0,Y 472.953,Z 277.572,A -85,B 0,C 180,E1 -5754.784,E2 -5754.784} C_VEL
LIN {X 0,Y 472.947,Z 277.573,A -85,B 0,C 180,E1 -5758.425,E2 -5758.425} C_VEL
LIN {X 0,Y 472.917,Z 277.573,A -85,B 0,C 180,E1 -5761.938,E2 -5761.938} C_VEL
LIN {X 0,Y 472.919,Z 277.573,A -85,B 0,C 180,E1 -5765.581,E2 -5765.581} C_VEL
LIN {X 0,Y 472.947,Z 277.567,A -85,B 0,C 180,E1 -5769.123,E2 -5769.123} C_VEL
LIN {X 0,Y 472.955,Z 277.57,A -85,B 0,C 180,E1 -5772.825,E2 -5772.825} C_VEL
LIN {X 0,Y 472.939,Z 277.572,A -85,B 0,C 180,E1 -5776.457,E2 -5776.457} C_VEL
LIN {X 0,Y 472.919,Z 277.573,A -85,B 0,C 180,E1 -5780.029,E2 -5780.029} C_VEL
LIN {X 0,Y 472.924,Z 277.573,A -85,B 0,C 180,E1 -5783.735,E2 -5783.735} C_VEL
LIN {X 0,Y 472.947,Z 277.569,A -85,B 0,C 180,E1 -5787.391,E2 -5787.391} C_VEL
LIN {X 0,Y 472.956,Z 277.571,A -85,B 0,C 180,E1 -5791.053,E2 -5791.053} C_VEL
LIN {X 0,Y 472.944,Z 277.574,A -85,B 0,C 180,E1 -5794.679,E2 -5794.679} C_VEL
LIN {X 0,Y 472.924,Z 277.573,A -85,B 0,C 180,E1 -5798.276,E2 -5798.276} C_VEL
LIN {X 0,Y 472.927,Z 277.574,A -85,B 0,C 180,E1 -5801.919,E2 -5801.919} C_VEL
LIN {X 0,Y 472.951,Z 277.572,A -85,B 0,C 180,E1 -5805.434,E2 -5805.434} C_VEL
LIN {X 0,Y 472.958,Z 277.574,A -85,B 0,C 180,E1 -5809.056,E2 -5809.056} C_VEL
LIN {X 0,Y 472.976,Z 277.929,A -85,B 0,C 180,E1 -5810.19,E2 -5810.19} C_VEL
LIN {X 0,Y 482.114,Z 300.518,A -85,B 0,C 180,E1 -5813.081,E2 -5813.081} C_VEL
LIN {X 0,Y 486.799,Z 313.699,A -85,B 0,C 180,E1 -5814.607,E2 -5814.607} C_VEL
LIN {X 0,Y 486.741,Z 317.483,A -85,B 0,C 180,E1 -5814.865,E2 -5814.865} C_VEL
LIN {X 0,Y 489.712,Z 338.32,A -85,B 0,C 180,E1 -5815.492,E2 -5815.492} C_VEL
LIN {X 0,Y 485.818,Z 547.216,A -85,B 0,C 180,E1 -5818.959,E2 -5818.959} C_VEL
LIN {X 0,Y 485.253,Z 578.797,A -85,B 0,C 180,E1 -5819.494,E2 -5819.494} C_VEL
LIN {X 0,Y 484.4,Z 599.834,A -85,B 0,C 180,E1 -5820.063,E2 -5820.063} C_VEL
LIN {X 0,Y 483.303,Z 621.042,A -85,B 0,C 180,E1 -5820.879,E2 -5820.879} C_VEL
LIN {X 0,Y 481.99,Z 641.435,A -85,B 0,C 180,E1 -5821.909,E2 -5821.909} C_VEL
LIN {X 0,Y 480.635,Z 660.241,A -85,B 0,C 180,E1 -5823.1,E2 -5823.1} C_VEL
LIN {X 0,Y 479.226,Z 678.232,A -85,B 0,C 180,E1 -5824.481,E2 -5824.481} C_VEL
LIN {X 0,Y 477.805,Z 695.344,A -85,B 0,C 180,E1 -5826.05,E2 -5826.05} C_VEL
LIN {X 0,Y 476.431,Z 711.863,A -85,B 0,C 180,E1 -5827.853,E2 -5827.853} C_VEL
LIN {X 0,Y 475.271,Z 726.138,A -85,B 0,C 180,E1 -5829.69,E2 -5829.69} C_VEL
LIN {X 0,Y 474.26,Z 739.363,A -85,B 0,C 180,E1 -5831.693,E2 -5831.693} C_VEL
LIN {X 0,Y 473.384,Z 751.826,A -85,B 0,C 180,E1 -5833.951,E2 -5833.951} C_VEL
LIN {X 0,Y 472.771,Z 761.962,A -85,B 0,C 180,E1 -5836.175,E2 -5836.175} C_VEL
LIN {X 0,Y 472.355,Z 770.304,A -85,B 0,C 180,E1 -5838.401,E2 -5838.401} C_VEL
LIN {X 0,Y 472.097,Z 777.293,A -85,B 0,C 180,E1 -5840.739,E2 -5840.739} C_VEL
LIN {X 0,Y 471.974,Z 782.512,A -85,B 0,C 180,E1 -5843.066,E2 -5843.066} C_VEL
LIN {X 0,Y 471.919,Z 786.247,A -85,B 0,C 180,E1 -5845.505,E2 -5845.505} C_VEL
LIN {X 0,Y 471.91,Z 788.371,A -85,B 0,C 180,E1 -5847.937,E2 -5847.937} C_VEL
LIN {X 0,Y 471.901,Z 788.916,A -85,B 0,C 180,E1 -5850.487,E2 -5850.487} C_VEL
LIN {X 0,Y 471.909,Z 787.843,A -85,B 0,C 180,E1 -5852.916,E2 -5852.916} C_VEL
LIN {X 0,Y 471.924,Z 785.124,A -85,B 0,C 180,E1 -5855.35,E2 -5855.35} C_VEL
LIN {X 0,Y 472.014,Z 780.732,A -85,B 0,C 180,E1 -5857.793,E2 -5857.793} C_VEL
LIN {X 0,Y 472.183,Z 774.94,A -85,B 0,C 180,E1 -5860.124,E2 -5860.124} C_VEL
LIN {X 0,Y 472.469,Z 767.71,A -85,B 0,C 180,E1 -5862.343,E2 -5862.343} C_VEL
LIN {X 0,Y 472.982,Z 758.094,A -85,B 0,C 180,E1 -5864.696,E2 -5864.696} C_VEL
LIN {X 0,Y 473.671,Z 746.862,A -85,B 0,C 180,E1 -5866.937,E2 -5866.937} C_VEL
LIN {X 0,Y 474.568,Z 734.047,A -85,B 0,C 180,E1 -5869.062,E2 -5869.062} C_VEL
LIN {X 0,Y 475.639,Z 719.598,A -85,B 0,C 180,E1 -5871.068,E2 -5871.068} C_VEL
LIN {X 0,Y 476.834,Z 703.931,A -85,B 0,C 180,E1 -5872.897,E2 -5872.897} C_VEL
LIN {X 0,Y 478.149,Z 686.621,A -85,B 0,C 180,E1 -5874.592,E2 -5874.592} C_VEL
LIN {X 0,Y 479.426,Z 668.869,A -85,B 0,C 180,E1 -5876.041,E2 -5876.041} C_VEL
LIN {X 0,Y 480.65,Z 650.205,A -85,B 0,C 180,E1 -5877.304,E2 -5877.304} C_VEL
LIN {X 0,Y 481.817,Z 630.66,A -85,B 0,C 180,E1 -5878.375,E2 -5878.375} C_VEL
LIN {X 0,Y 482.816,Z 610.013,A -85,B 0,C 180,E1 -5879.258,E2 -5879.258} C_VEL
LIN {X 0,Y 483.647,Z 588.937,A -85,B 0,C 180,E1 -5879.922,E2 -5879.922} C_VEL
LIN {X 0,Y 484.197,Z 567.797,A -85,B 0,C 180,E1 -5880.367,E2 -5880.367} C_VEL
LIN {X 0,Y 486.013,Z 442.58,A -85,B 0,C 180,E1 -5882.388,E2 -5882.388} C_VEL
LIN {X 0,Y 488.48,Z 339.694,A -85,B 0,C 180,E1 -5884.245,E2 -5884.245} C_VEL
LIN {X 0,Y 488.291,Z 334.925,A -85,B 0,C 180,E1 -5884.362,E2 -5884.362} C_VEL
LIN {X 0,Y 486.291,Z 319.701,A -85,B 0,C 180,E1 -5884.878,E2 -5884.878} C_VEL
LIN {X 0,Y 486.684,Z 312.859,A -85,B 0,C 180,E1 -5885.454,E2 -5885.454} C_VEL
LIN {X 0,Y 482.508,Z 299.812,A -85,B 0,C 180,E1 -5887.188,E2 -5887.188} C_VEL
LIN {X 0,Y 478.669,Z 289.95,A -85,B 0,C 180,E1 -5888.819,E2 -5888.819} C_VEL
LIN {X 0,Y 476.698,Z 285.829,A -85,B 0,C 180,E1 -5889.667,E2 -5889.667} C_VEL
LIN {X 0,Y 474.868,Z 281.861,A -85,B 0,C 180,E1 -5890.589,E2 -5890.589} C_VEL
LIN {X 0,Y 473,Z 278.092,A -85,B 0,C 180,E1 -5891.683,E2 -5891.683} C_VEL
LIN {X 0,Y 472.946,Z 277.575,A -85,B 0,C 180,E1 -5892.409,E2 -5892.409} C_VEL
LIN {X 0,Y 472.919,Z 277.579,A -85,B 0,C 180,E1 -5895.96,E2 -5895.96} C_VEL
LIN {X 0,Y 472.918,Z 277.579,A -85,B 0,C 180,E1 -5899.564,E2 -5899.564} C_VEL
LIN {X 0,Y 473.012,Z 278.109,A -85,B 0,C 180,E1 -5900.251,E2 -5900.251} C_VEL
LIN {X 0,Y 474.946,Z 282.011,A -85,B 0,C 180,E1 -5901.455,E2 -5901.455} C_VEL
LIN {X 0,Y 477.472,Z 287.685,A -85,B 0,C 180,E1 -5902.826,E2 -5902.826} C_VEL
LIN {X 0,Y 480.774,Z 295.609,A -85,B 0,C 180,E1 -5904.407,E2 -5904.407} C_VEL
LIN {X 0,Y 484.37,Z 306.095,A -85,B 0,C 180,E1 -5906.128,E2 -5906.128} C_VEL
LIN {X 0,Y 486.032,Z 311.9,A -85,B 0,C 180,E1 -5906.965,E2 -5906.965} C_VEL
LIN {X 0,Y 483.594,Z 340.076,A -85,B 0,C 180,E1 -5909.674,E2 -5909.674} C_VEL
LIN {X 0,Y 487.001,Z 362.667,A -85,B 0,C 180,E1 -5910.523,E2 -5910.523} C_VEL
LIN {X 0,Y 484.009,Z 460.793,A -85,B 0,C 180,E1 -5912.367,E2 -5912.367} C_VEL
LIN {X 0,Y 481.994,Z 563.137,A -85,B 0,C 180,E1 -5914.154,E2 -5914.154} C_VEL
LIN {X 0,Y 481.292,Z 582.634,A -85,B 0,C 180,E1 -5914.712,E2 -5914.712} C_VEL
LIN {X 0,Y 480.419,Z 601.195,A -85,B 0,C 180,E1 -5915.462,E2 -5915.462} C_VEL
LIN {X 0,Y 479.428,Z 618.87,A -85,B 0,C 180,E1 -5916.396,E2 -5916.396} C_VEL
LIN {X 0,Y 478.335,Z 635.688,A -85,B 0,C 180,E1 -5917.51,E2 -5917.51} C_VEL
LIN {X 0,Y 477.193,Z 651.709,A -85,B 0,C 180,E1 -5918.814,E2 -5918.814} C_VEL
LIN {X 0,Y 476.057,Z 666.755,A -85,B 0,C 180,E1 -5920.3,E2 -5920.3} C_VEL
LIN {X 0,Y 474.979,Z 680.816,A -85,B 0,C 180,E1 -5921.975,E2 -5921.975} C_VEL
LIN {X 0,Y 474.079,Z 692.989,A -85,B 0,C 180,E1 -5923.71,E2 -5923.71} C_VEL
LIN {X 0,Y 473.281,Z 704.442,A -85,B 0,C 180,E1 -5925.69,E2 -5925.69} C_VEL
LIN {X 0,Y 472.682,Z 714.316,A -85,B 0,C 180,E1 -5927.788,E2 -5927.788} C_VEL
LIN {X 0,Y 472.273,Z 722.646,A -85,B 0,C 180,E1 -5930.003,E2 -5930.003} C_VEL
LIN {X 0,Y 472.049,Z 729.142,A -85,B 0,C 180,E1 -5932.209,E2 -5932.209} C_VEL
LIN {X 0,Y 471.95,Z 733.915,A -85,B 0,C 180,E1 -5934.408,E2 -5934.408} C_VEL
LIN {X 0,Y 471.916,Z 737.192,A -85,B 0,C 180,E1 -5936.721,E2 -5936.721} C_VEL
LIN {X 0,Y 471.916,Z 738.794,A -85,B 0,C 180,E1 -5939.029,E2 -5939.029} C_VEL
LIN {X 0,Y 471.911,Z 738.735,A -85,B 0,C 180,E1 -5941.336,E2 -5941.336} C_VEL
LIN {X 0,Y 471.914,Z 737.031,A -85,B 0,C 180,E1 -5943.523,E2 -5943.523} C_VEL
LIN {X 0,Y 471.953,Z 733.614,A -85,B 0,C 180,E1 -5945.837,E2 -5945.837} C_VEL
LIN {X 0,Y 472.062,Z 728.762,A -85,B 0,C 180,E1 -5948.036,E2 -5948.036} C_VEL
LIN {X 0,Y 472.311,Z 721.725,A -85,B 0,C 180,E1 -5950.367,E2 -5950.367} C_VEL
LIN {X 0,Y 472.711,Z 713.596,A -85,B 0,C 180,E1 -5952.46,E2 -5952.46} C_VEL
LIN {X 0,Y 473.328,Z 703.509,A -85,B 0,C 180,E1 -5954.559,E2 -5954.559} C_VEL
LIN {X 0,Y 474.146,Z 691.867,A -85,B 0,C 180,E1 -5956.54,E2 -5956.54} C_VEL
LIN {X 0,Y 475.156,Z 678.618,A -85,B 0,C 180,E1 -5958.4,E2 -5958.4} C_VEL
LIN {X 0,Y 476.271,Z 664.265,A -85,B 0,C 180,E1 -5960.066,E2 -5960.066} C_VEL
LIN {X 0,Y 477.513,Z 648.11,A -85,B 0,C 180,E1 -5961.612,E2 -5961.612} C_VEL
LIN {X 0,Y 478.711,Z 631.572,A -85,B 0,C 180,E1 -5962.912,E2 -5962.912} C_VEL
LIN {X 0,Y 479.878,Z 613.747,A -85,B 0,C 180,E1 -5964.038,E2 -5964.038} C_VEL
LIN {X 0,Y 480.911,Z 595.779,A -85,B 0,C 180,E1 -5964.932,E2 -5964.932} C_VEL
LIN {X 0,Y 481.785,Z 576.374,A -85,B 0,C 180,E1 -5965.652,E2 -5965.652} C_VEL
LIN {X 0,Y 482.432,Z 556.759,A -85,B 0,C 180,E1 -5966.143,E2 -5966.143} C_VEL
LIN {X 0,Y 485.739,Z 361.781,A -85,B 0,C 180,E1 -5969.362,E2 -5969.362} C_VEL
LIN {X 0,Y 482.407,Z 341.183,A -85,B 0,C 180,E1 -5970.003,E2 -5970.003} C_VEL
LIN {X 0,Y 484.309,Z 309.352,A -85,B 0,C 180,E1 -5972.93,E2 -5972.93} C_VEL
LIN {X 0,Y 481.268,Z 300.303,A -85,B 0,C 180,E1 -5974.072,E2 -5974.072} C_VEL
LIN {X 0,Y 479.033,Z 296.363,A -85,B 0,C 180,E1 -5974.656,E2 -5974.656} C_VEL
LIN {X 0,Y 472.411,Z 290.224,A -85,B 0,C 180,E1 -5975.861,E2 -5975.861} C_VEL
LIN {X 0,Y 467.825,Z 285.382,A -85,B 0,C 180,E1 -5976.782,E2 -5976.782} C_VEL
LIN {X 0,Y 466.245,Z 281.995,A -85,B 0,C 180,E1 -5977.285,E2 -5977.285} C_VEL
LIN {X 0,Y 465.013,Z 278.744,A -85,B 0,C 180,E1 -5977.81,E2 -5977.81} C_VEL
LIN {X 0,Y 465.017,Z 278.556,A -85,B 0,C 180,E1 -5981.373,E2 -5981.373} C_VEL
LIN {X 0,Y 465.012,Z 278.562,A -85,B 0,C 180,E1 -5985.025,E2 -5985.025} C_VEL
LIN {X 0,Y 465.015,Z 278.563,A -85,B 0,C 180,E1 -5988.691,E2 -5988.691} C_VEL
LIN {X 0,Y 465.009,Z 278.563,A -85,B 0,C 180,E1 -5992.362,E2 -5992.362} C_VEL
LIN {X 0,Y 465.01,Z 278.561,A -85,B 0,C 180,E1 -5996.097,E2 -5996.097} C_VEL
LIN {X 0,Y 465.019,Z 278.553,A -85,B 0,C 180,E1 -5999.811,E2 -5999.811} C_VEL
LIN {X 0,Y 464.996,Z 278.561,A -85,B 0,C 180,E1 -6003.446,E2 -6003.446} C_VEL
LIN {X 0,Y 464.979,Z 278.564,A -85,B 0,C 180,E1 -6007.094,E2 -6007.094} C_VEL
LIN {X 0,Y 464.971,Z 278.565,A -85,B 0,C 180,E1 -6010.79,E2 -6010.79} C_VEL
LIN {X 0,Y 464.979,Z 278.549,A -85,B 0,C 180,E1 -6014.406,E2 -6014.406} C_VEL
LIN {X 0,Y 464.982,Z 278.766,A -85,B 0,C 180,E1 -6016.887,E2 -6016.887} C_VEL
LIN {X 0,Y 466.456,Z 283.117,A -85,B 0,C 180,E1 -6017.433,E2 -6017.433} C_VEL
LIN {X 0,Y 473.182,Z 302.832,A -85,B 0,C 180,E1 -6019.652,E2 -6019.652} C_VEL
LIN {X 0,Y 474.745,Z 308.341,A -85,B 0,C 180,E1 -6020.238,E2 -6020.238} C_VEL
LIN {X 0,Y 473.565,Z 350.556,A -85,B 0,C 180,E1 -6023.817,E2 -6023.817} C_VEL
LIN {X 0,Y 472.253,Z 392.103,A -85,B 0,C 180,E1 -6027.329,E2 -6027.329} C_VEL
LIN {X 0,Y 470.814,Z 432.969,A -85,B 0,C 180,E1 -6030.79,E2 -6030.79} C_VEL
LIN {X 0,Y 469.546,Z 472.848,A -85,B 0,C 180,E1 -6034.15,E2 -6034.15} C_VEL
LIN {X 0,Y 469.578,Z 476.566,A -85,B 0,C 180,E1 -6034.403,E2 -6034.403} C_VEL
LIN {X 0,Y 470.822,Z 489.015,A -85,B 0,C 180,E1 -6034.66,E2 -6034.66} C_VEL
LIN {X 0,Y 469.449,Z 618.878,A -85,B 0,C 180,E1 -6036.707,E2 -6036.707} C_VEL
LIN {X 0,Y 469.082,Z 634.851,A -85,B 0,C 180,E1 -6037.183,E2 -6037.183} C_VEL
LIN {X 0,Y 468.512,Z 651.058,A -85,B 0,C 180,E1 -6037.911,E2 -6037.911} C_VEL
LIN {X 0,Y 467.845,Z 665.454,A -85,B 0,C 180,E1 -6038.794,E2 -6038.794} C_VEL
LIN {X 0,Y 467.072,Z 679.637,A -85,B 0,C 180,E1 -6039.922,E2 -6039.922} C_VEL
LIN {X 0,Y 466.353,Z 692.226,A -85,B 0,C 180,E1 -6041.187,E2 -6041.187} C_VEL
LIN {X 0,Y 465.652,Z 703.866,A -85,B 0,C 180,E1 -6042.65,E2 -6042.65} C_VEL
LIN {X 0,Y 465.089,Z 713.732,A -85,B 0,C 180,E1 -6044.185,E2 -6044.185} C_VEL
LIN {X 0,Y 464.603,Z 722.84,A -85,B 0,C 180,E1 -6045.988,E2 -6045.988} C_VEL
LIN {X 0,Y 464.291,Z 730.112,A -85,B 0,C 180,E1 -6047.849,E2 -6047.849} C_VEL
LIN {X 0,Y 464.104,Z 735.561,A -85,B 0,C 180,E1 -6049.768,E2 -6049.768} C_VEL
LIN {X 0,Y 464.018,Z 739.387,A -85,B 0,C 180,E1 -6051.763,E2 -6051.763} C_VEL
LIN {X 0,Y 463.985,Z 741.358,A -85,B 0,C 180,E1 -6053.762,E2 -6053.762} C_VEL
LIN {X 0,Y 463.985,Z 741.633,A -85,B 0,C 180,E1 -6055.802,E2 -6055.802} C_VEL
LIN {X 0,Y 464.005,Z 740.18,A -85,B 0,C 180,E1 -6057.737,E2 -6057.737} C_VEL
LIN {X 0,Y 464.083,Z 736.734,A -85,B 0,C 180,E1 -6059.845,E2 -6059.845} C_VEL
LIN {X 0,Y 464.234,Z 731.911,A -85,B 0,C 180,E1 -6061.706,E2 -6061.706} C_VEL
LIN {X 0,Y 464.513,Z 725.176,A -85,B 0,C 180,E1 -6063.589,E2 -6063.589} C_VEL
LIN {X 0,Y 464.932,Z 716.977,A -85,B 0,C 180,E1 -6065.343,E2 -6065.343} C_VEL
LIN {X 0,Y 465.541,Z 706.308,A -85,B 0,C 180,E1 -6067.12,E2 -6067.12} C_VEL
LIN {X 0,Y 466.222,Z 694.964,A -85,B 0,C 180,E1 -6068.612,E2 -6068.612} C_VEL
LIN {X 0,Y 466.976,Z 682.126,A -85,B 0,C 180,E1 -6069.964,E2 -6069.964} C_VEL
LIN {X 0,Y 467.727,Z 668.425,A -85,B 0,C 180,E1 -6071.102,E2 -6071.102} C_VEL
LIN {X 0,Y 468.461,Z 653.228,A -85,B 0,C 180,E1 -6072.079,E2 -6072.079} C_VEL
LIN {X 0,Y 469.026,Z 637.742,A -85,B 0,C 180,E1 -6072.809,E2 -6072.809} C_VEL
LIN {X 0,Y 469.43,Z 621.065,A -85,B 0,C 180,E1 -6073.344,E2 -6073.344} C_VEL
LIN {X 0,Y 469.75,Z 591.011,A -85,B 0,C 180,E1 -6073.856,E2 -6073.856} C_VEL
LIN {X 0,Y 470.685,Z 485.447,A -85,B 0,C 180,E1 -6075.513,E2 -6075.513} C_VEL
LIN {X 0,Y 469.532,Z 475.788,A -85,B 0,C 180,E1 -6075.742,E2 -6075.742} C_VEL
LIN {X 0,Y 470.835,Z 433.125,A -85,B 0,C 180,E1 -6079.311,E2 -6079.311} C_VEL
LIN {X 0,Y 472.249,Z 391.324,A -85,B 0,C 180,E1 -6082.809,E2 -6082.809} C_VEL
LIN {X 0,Y 473.35,Z 347.842,A -85,B 0,C 180,E1 -6086.397,E2 -6086.397} C_VEL
LIN {X 0,Y 474.148,Z 309.128,A -85,B 0,C 180,E1 -6089.595,E2 -6089.595} C_VEL
LIN {X 0,Y 473.942,Z 305.321,A -85,B 0,C 180,E1 -6089.93,E2 -6089.93} C_VEL
LIN {X 0,Y 467.735,Z 286.545,A -85,B 0,C 180,E1 -6091.947,E2 -6091.947} C_VEL
LIN {X 0,Y 465.04,Z 278.849,A -85,B 0,C 180,E1 -6092.848,E2 -6092.848} C_VEL
LIN {X 0,Y 465.014,Z 278.559,A -85,B 0,C 180,E1 -6094.56,E2 -6094.56} C_VEL
LIN {X 0,Y 465.011,Z 278.56,A -85,B 0,C 180,E1 -6098.255,E2 -6098.255} C_VEL
LIN {X 0,Y 464.981,Z 278.559,A -85,B 0,C 180,E1 -6101.88,E2 -6101.88} C_VEL
LIN {X 0,Y 464.973,Z 278.563,A -85,B 0,C 180,E1 -6105.555,E2 -6105.555} C_VEL
LIN {X 0,Y 464.987,Z 278.561,A -85,B 0,C 180,E1 -6109.217,E2 -6109.217} C_VEL
LIN {X 0,Y 465.019,Z 278.559,A -85,B 0,C 180,E1 -6112.836,E2 -6112.836} C_VEL
LIN {X 0,Y 465.012,Z 278.562,A -85,B 0,C 180,E1 -6116.548,E2 -6116.548} C_VEL
LIN {X 0,Y 464.987,Z 278.565,A -85,B 0,C 180,E1 -6120.123,E2 -6120.123} C_VEL
LIN {X 0,Y 464.977,Z 278.561,A -85,B 0,C 180,E1 -6123.698,E2 -6123.698} C_VEL
LIN {X 0,Y 464.998,Z 278.559,A -85,B 0,C 180,E1 -6127.288,E2 -6127.288} C_VEL
LIN {X 0,Y 465.014,Z 278.561,A -85,B 0,C 180,E1 -6130.907,E2 -6130.907} C_VEL
LIN {X 0,Y 465.016,Z 278.562,A -85,B 0,C 180,E1 -6134.639,E2 -6134.639} C_VEL
LIN {X 0,Y 464.99,Z 278.565,A -85,B 0,C 180,E1 -6138.296,E2 -6138.296} C_VEL
LIN {X 0,Y 464.979,Z 278.56,A -85,B 0,C 180,E1 -6141.972,E2 -6141.972} C_VEL
LIN {X 0,Y 464.992,Z 278.561,A -85,B 0,C 180,E1 -6145.607,E2 -6145.607} C_VEL
LIN {X 0,Y 465.019,Z 278.557,A -85,B 0,C 180,E1 -6149.214,E2 -6149.214} C_VEL
LIN {X 0,Y 465.016,Z 278.563,A -85,B 0,C 180,E1 -6152.955,E2 -6152.955} C_VEL
LIN {X 0,Y 465.004,Z 278.563,A -85,B 0,C 180,E1 -6156.679,E2 -6156.679} C_VEL
LIN {X 0,Y 464.986,Z 278.563,A -85,B 0,C 180,E1 -6160.242,E2 -6160.242} C_VEL
LIN {X 0,Y 464.989,Z 278.565,A -85,B 0,C 180,E1 -6163.99,E2 -6163.99} C_VEL
LIN {X 0,Y 465.01,Z 278.562,A -85,B 0,C 180,E1 -6167.536,E2 -6167.536} C_VEL
LIN {X 0,Y 465.058,Z 278.859,A -85,B 0,C 180,E1 -6169.514,E2 -6169.514} C_VEL
LIN {X 0,Y 474.564,Z 302.305,A -85,B 0,C 180,E1 -6172.589,E2 -6172.589} C_VEL
LIN {X 0,Y 479.76,Z 316.657,A -85,B 0,C 180,E1 -6174.284,E2 -6174.284} C_VEL
LIN {X 0,Y 482.961,Z 339.639,A -85,B 0,C 180,E1 -6175.001,E2 -6175.001} C_VEL
LIN {X 0,Y 478.751,Z 545.861,A -85,B 0,C 180,E1 -6178.495,E2 -6178.495} C_VEL
LIN {X 0,Y 478.071,Z 579.185,A -85,B 0,C 180,E1 -6179.078,E2 -6179.078} C_VEL
LIN {X 0,Y 477.16,Z 600.106,A -85,B 0,C 180,E1 -6179.658,E2 -6179.658} C_VEL
LIN {X 0,Y 476.027,Z 620.636,A -85,B 0,C 180,E1 -6180.459,E2 -6180.459} C_VEL
LIN {X 0,Y 474.706,Z 639.892,A -85,B 0,C 180,E1 -6181.439,E2 -6181.439} C_VEL
LIN {X 0,Y 473.292,Z 658.653,A -85,B 0,C 180,E1 -6182.626,E2 -6182.626} C_VEL
LIN {X 0,Y 471.748,Z 677.12,A -85,B 0,C 180,E1 -6184.046,E2 -6184.046} C_VEL
LIN {X 0,Y 470.177,Z 695.002,A -85,B 0,C 180,E1 -6185.703,E2 -6185.703} C_VEL
LIN {X 0,Y 468.783,Z 710.825,A -85,B 0,C 180,E1 -6187.448,E2 -6187.448} C_VEL
LIN {X 0,Y 467.514,Z 725.381,A -85,B 0,C 180,E1 -6189.338,E2 -6189.338} C_VEL
LIN {X 0,Y 466.423,Z 738.67,A -85,B 0,C 180,E1 -6191.375,E2 -6191.375} C_VEL
LIN {X 0,Y 465.488,Z 751.127,A -85,B 0,C 180,E1 -6193.659,E2 -6193.659} C_VEL
LIN {X 0,Y 464.82,Z 761.497,A -85,B 0,C 180,E1 -6195.96,E2 -6195.96} C_VEL
LIN {X 0,Y 464.368,Z 770.2,A -85,B 0,C 180,E1 -6198.324,E2 -6198.324} C_VEL
LIN {X 0,Y 464.092,Z 777.478,A -85,B 0,C 180,E1 -6200.828,E2 -6200.828} C_VEL
LIN {X 0,Y 463.973,Z 782.678,A -85,B 0,C 180,E1 -6203.194,E2 -6203.194} C_VEL
LIN {X 0,Y 463.918,Z 786.418,A -85,B 0,C 180,E1 -6205.675,E2 -6205.675} C_VEL
LIN {X 0,Y 463.91,Z 788.349,A -85,B 0,C 180,E1 -6208.025,E2 -6208.025} C_VEL
LIN {X 0,Y 463.901,Z 788.838,A -85,B 0,C 180,E1 -6210.495,E2 -6210.495} C_VEL
LIN {X 0,Y 463.908,Z 787.729,A -85,B 0,C 180,E1 -6212.966,E2 -6212.966} C_VEL
LIN {X 0,Y 463.926,Z 784.921,A -85,B 0,C 180,E1 -6215.443,E2 -6215.443} C_VEL
LIN {X 0,Y 464.015,Z 780.63,A -85,B 0,C 180,E1 -6217.803,E2 -6217.803} C_VEL
LIN {X 0,Y 464.202,Z 774.354,A -85,B 0,C 180,E1 -6220.3,E2 -6220.3} C_VEL
LIN {X 0,Y 464.53,Z 766.554,A -85,B 0,C 180,E1 -6222.684,E2 -6222.684} C_VEL
LIN {X 0,Y 465.051,Z 757.327,A -85,B 0,C 180,E1 -6224.953,E2 -6224.953} C_VEL
LIN {X 0,Y 465.784,Z 745.968,A -85,B 0,C 180,E1 -6227.233,E2 -6227.233} C_VEL
LIN {X 0,Y 466.676,Z 733.824,A -85,B 0,C 180,E1 -6229.267,E2 -6229.267} C_VEL
LIN {X 0,Y 467.804,Z 719.357,A -85,B 0,C 180,E1 -6231.307,E2 -6231.307} C_VEL
LIN {X 0,Y 469.049,Z 703.761,A -85,B 0,C 180,E1 -6233.156,E2 -6233.156} C_VEL
LIN {X 0,Y 470.382,Z 687.086,A -85,B 0,C 180,E1 -6234.819,E2 -6234.819} C_VEL
LIN {X 0,Y 471.67,Z 670.168,A -85,B 0,C 180,E1 -6236.238,E2 -6236.238} C_VEL
LIN {X 0,Y 473.009,Z 650.857,A -85,B 0,C 180,E1 -6237.577,E2 -6237.577} C_VEL
LIN {X 0,Y 474.238,Z 631.347,A -85,B 0,C 180,E1 -6238.67,E2 -6238.67} C_VEL
LIN {X 0,Y 475.289,Z 611.052,A -85,B 0,C 180,E1 -6239.565,E2 -6239.565} C_VEL
LIN {X 0,Y 476.177,Z 590.629,A -85,B 0,C 180,E1 -6240.236,E2 -6240.236} C_VEL
LIN {X 0,Y 476.804,Z 569.324,A -85,B 0,C 180,E1 -6240.716,E2 -6240.716} C_VEL
LIN {X 0,Y 478.808,Z 448.931,A -85,B 0,C 180,E1 -6242.725,E2 -6242.725} C_VEL
LIN {X 0,Y 481.529,Z 349.387,A -85,B 0,C 180,E1 -6244.587,E2 -6244.587} C_VEL
LIN {X 0,Y 481.755,Z 336.867,A -85,B 0,C 180,E1 -6244.857,E2 -6244.857} C_VEL
LIN {X 0,Y 479.668,Z 320.237,A -85,B 0,C 180,E1 -6245.452,E2 -6245.452} C_VEL
LIN {X 0,Y 479.84,Z 315.899,A -85,B 0,C 180,E1 -6245.849,E2 -6245.849} C_VEL
LIN {X 0,Y 476.154,Z 303.9,A -85,B 0,C 180,E1 -6247.515,E2 -6247.515} C_VEL
LIN {X 0,Y 472.733,Z 294.953,A -85,B 0,C 180,E1 -6249.084,E2 -6249.084} C_VEL
LIN {X 0,Y 470.866,Z 290.962,A -85,B 0,C 180,E1 -6249.954,E2 -6249.954} C_VEL
LIN {X 0,Y 469.248,Z 287.348,A -85,B 0,C 180,E1 -6250.851,E2 -6250.851} C_VEL
LIN {X 0,Y 467.388,Z 283.398,A -85,B 0,C 180,E1 -6252.071,E2 -6252.071} C_VEL
LIN {X 0,Y 465.308,Z 280.047,A -85,B 0,C 180,E1 -6253.783,E2 -6253.783} C_VEL
LIN {X 0,Y 465.034,Z 278.718,A -85,B 0,C 180,E1 -6254.93,E2 -6254.93} C_VEL
LIN {X 0,Y 465.049,Z 278.954,A -85,B 0,C 180,E1 -6257.334,E2 -6257.334} C_VEL
LIN {X 0,Y 466.072,Z 281.646,A -85,B 0,C 180,E1 -6258.97,E2 -6258.97} C_VEL
LIN {X 0,Y 467.702,Z 284.057,A -85,B 0,C 180,E1 -6260.129,E2 -6260.129} C_VEL
LIN {X 0,Y 469.858,Z 288.793,A -85,B 0,C 180,E1 -6261.584,E2 -6261.584} C_VEL
LIN {X 0,Y 471.799,Z 293.272,A -85,B 0,C 180,E1 -6262.692,E2 -6262.692} C_VEL
LIN {X 0,Y 475.156,Z 301.73,A -85,B 0,C 180,E1 -6264.421,E2 -6264.421} C_VEL
LIN {X 0,Y 478.806,Z 313.207,A -85,B 0,C 180,E1 -6266.312,E2 -6266.312} C_VEL
LIN {X 0,Y 479.261,Z 315.658,A -85,B 0,C 180,E1 -6266.652,E2 -6266.652} C_VEL
LIN {X 0,Y 476.918,Z 339.639,A -85,B 0,C 180,E1 -6269.011,E2 -6269.011} C_VEL
LIN {X 0,Y 480.174,Z 361.469,A -85,B 0,C 180,E1 -6269.899,E2 -6269.899} C_VEL
LIN {X 0,Y 480.378,Z 366.22,A -85,B 0,C 180,E1 -6270.035,E2 -6270.035} C_VEL
LIN {X 0,Y 477.019,Z 460.537,A -85,B 0,C 180,E1 -6271.898,E2 -6271.898} C_VEL
LIN {X 0,Y 474.641,Z 563.657,A -85,B 0,C 180,E1 -6273.782,E2 -6273.782} C_VEL
LIN {X 0,Y 473.877,Z 583.372,A -85,B 0,C 180,E1 -6274.362,E2 -6274.362} C_VEL
LIN {X 0,Y 472.956,Z 601.758,A -85,B 0,C 180,E1 -6275.122,E2 -6275.122} C_VEL
LIN {X 0,Y 471.847,Z 620.292,A -85,B 0,C 180,E1 -6276.126,E2 -6276.126} C_VEL
LIN {X 0,Y 470.644,Z 637.749,A -85,B 0,C 180,E1 -6277.32,E2 -6277.32} C_VEL
LIN {X 0,Y 469.401,Z 654.23,A -85,B 0,C 180,E1 -6278.711,E2 -6278.711} C_VEL
LIN {X 0,Y 468.177,Z 669.503,A -85,B 0,C 180,E1 -6280.28,E2 -6280.28} C_VEL
LIN {X 0,Y 467.107,Z 682.742,A -85,B 0,C 180,E1 -6281.918,E2 -6281.918} C_VEL
LIN {X 0,Y 466.111,Z 695.456,A -85,B 0,C 180,E1 -6283.808,E2 -6283.808} C_VEL
LIN {X 0,Y 465.303,Z 706.599,A -85,B 0,C 180,E1 -6285.821,E2 -6285.821} C_VEL
LIN {X 0,Y 464.7,Z 716.19,A -85,B 0,C 180,E1 -6287.954,E2 -6287.954} C_VEL
LIN {X 0,Y 464.305,Z 723.807,A -85,B 0,C 180,E1 -6290.08,E2 -6290.08} C_VEL
LIN {X 0,Y 464.061,Z 730.154,A -85,B 0,C 180,E1 -6292.358,E2 -6292.358} C_VEL
LIN {X 0,Y 463.956,Z 734.835,A -85,B 0,C 180,E1 -6294.683,E2 -6294.683} C_VEL
LIN {X 0,Y 463.918,Z 737.769,A -85,B 0,C 180,E1 -6297.035,E2 -6297.035} C_VEL
LIN {X 0,Y 463.913,Z 739.024,A -85,B 0,C 180,E1 -6299.383,E2 -6299.383} C_VEL
LIN {X 0,Y 463.909,Z 738.679,A -85,B 0,C 180,E1 -6301.73,E2 -6301.73} C_VEL
LIN {X 0,Y 463.924,Z 736.7,A -85,B 0,C 180,E1 -6304.079,E2 -6304.079} C_VEL
LIN {X 0,Y 463.984,Z 732.925,A -85,B 0,C 180,E1 -6306.434,E2 -6306.434} C_VEL
LIN {X 0,Y 464.132,Z 727.681,A -85,B 0,C 180,E1 -6308.674,E2 -6308.674} C_VEL
LIN {X 0,Y 464.44,Z 720.672,A -85,B 0,C 180,E1 -6310.921,E2 -6310.921} C_VEL
LIN {X 0,Y 464.918,Z 712.234,A -85,B 0,C 180,E1 -6313.051,E2 -6313.051} C_VEL
LIN {X 0,Y 465.629,Z 701.682,A -85,B 0,C 180,E1 -6315.188,E2 -6315.188} C_VEL
LIN {X 0,Y 466.556,Z 689.485,A -85,B 0,C 180,E1 -6317.203,E2 -6317.203} C_VEL
LIN {X 0,Y 467.64,Z 676.063,A -85,B 0,C 180,E1 -6319.03,E2 -6319.03} C_VEL
LIN {X 0,Y 468.845,Z 661.674,A -85,B 0,C 180,E1 -6320.668,E2 -6320.668} C_VEL
LIN {X 0,Y 470.132,Z 645.791,A -85,B 0,C 180,E1 -6322.162,E2 -6322.162} C_VEL
LIN {X 0,Y 471.459,Z 628.384,A -85,B 0,C 180,E1 -6323.498,E2 -6323.498} C_VEL
LIN {X 0,Y 472.634,Z 611.107,A -85,B 0,C 180,E1 -6324.564,E2 -6324.564} C_VEL
LIN {X 0,Y 473.734,Z 592.303,A -85,B 0,C 180,E1 -6325.47,E2 -6325.47} C_VEL
LIN {X 0,Y 474.625,Z 573.24,A -85,B 0,C 180,E1 -6326.146,E2 -6326.146} C_VEL
LIN {X 0,Y 475.261,Z 553.681,A -85,B 0,C 180,E1 -6326.608,E2 -6326.608} C_VEL
LIN {X 0,Y 478.82,Z 362.881,A -85,B 0,C 180,E1 -6329.835,E2 -6329.835} C_VEL
LIN {X 0,Y 475.289,Z 340.988,A -85,B 0,C 180,E1 -6330.534,E2 -6330.534} C_VEL
LIN {X 0,Y 477.161,Z 312.369,A -85,B 0,C 180,E1 -6333.203,E2 -6333.203} C_VEL
LIN {X 0,Y 470.474,Z 293.202,A -85,B 0,C 180,E1 -6335.723,E2 -6335.723} C_VEL
LIN {X 0,Y 466.245,Z 281.995,A -85,B 0,C 180,E1 -6337.285,E2 -6337.285} C_VEL
LIN {X 0,Y 465.187,Z 279.902,A -85,B 0,C 180,E1 -6337.713,E2 -6337.713} C_VEL
LIN {X 0,Y 463.248,Z 278.89,A -85,B 0,C 180,E1 -6338.39,E2 -6338.39} C_VEL
LIN {X 0,Y 458.095,Z 279.463,A -85,B 0,C 180,E1 -6340.432,E2 -6340.432} C_VEL
LIN {X 0,Y 457.07,Z 279.544,A -85,B 0,C 180,E1 -6341.525,E2 -6341.525} C_VEL
LIN {X 0,Y 457.075,Z 279.552,A -85,B 0,C 180,E1 -6345.219,E2 -6345.219} C_VEL
LIN {X 0,Y 457.07,Z 279.552,A -85,B 0,C 180,E1 -6349,E2 -6349} C_VEL
LIN {X 0,Y 457.071,Z 279.553,A -85,B 0,C 180,E1 -6352.702,E2 -6352.702} C_VEL
LIN {X 0,Y 457.075,Z 279.553,A -85,B 0,C 180,E1 -6356.455,E2 -6356.455} C_VEL
LIN {X 0,Y 457.076,Z 279.537,A -85,B 0,C 180,E1 -6360.226,E2 -6360.226} C_VEL
LIN {X 0,Y 457.077,Z 279.547,A -85,B 0,C 180,E1 -6363.915,E2 -6363.915} C_VEL
LIN {X 0,Y 457.063,Z 279.552,A -85,B 0,C 180,E1 -6367.626,E2 -6367.626} C_VEL
LIN {X 0,Y 457.034,Z 279.551,A -85,B 0,C 180,E1 -6371.239,E2 -6371.239} C_VEL
LIN {X 0,Y 457.015,Z 279.526,A -85,B 0,C 180,E1 -6374.908,E2 -6374.908} C_VEL
LIN {X 0,Y 457.061,Z 279.687,A -85,B 0,C 180,E1 -6376.333,E2 -6376.333} C_VEL
LIN {X 0,Y 457.527,Z 281.498,A -85,B 0,C 180,E1 -6376.605,E2 -6376.605} C_VEL
LIN {X 0,Y 464.169,Z 299.981,A -85,B 0,C 180,E1 -6378.757,E2 -6378.757} C_VEL
LIN {X 0,Y 467.468,Z 310.94,A -85,B 0,C 180,E1 -6379.96,E2 -6379.96} C_VEL
LIN {X 0,Y 466.22,Z 351.998,A -85,B 0,C 180,E1 -6383.472,E2 -6383.472} C_VEL
LIN {X 0,Y 464.811,Z 393.857,A -85,B 0,C 180,E1 -6387.039,E2 -6387.039} C_VEL
LIN {X 0,Y 463.265,Z 435.826,A -85,B 0,C 180,E1 -6390.617,E2 -6390.617} C_VEL
LIN {X 0,Y 461.963,Z 476.377,A -85,B 0,C 180,E1 -6394.039,E2 -6394.039} C_VEL
LIN {X 0,Y 463.322,Z 489.694,A -85,B 0,C 180,E1 -6394.325,E2 -6394.325} C_VEL
LIN {X 0,Y 461.853,Z 619.179,A -85,B 0,C 180,E1 -6396.4,E2 -6396.4} C_VEL
LIN {X 0,Y 461.468,Z 635.14,A -85,B 0,C 180,E1 -6396.882,E2 -6396.882} C_VEL
LIN {X 0,Y 460.877,Z 651.033,A -85,B 0,C 180,E1 -6397.603,E2 -6397.603} C_VEL
LIN {X 0,Y 460.175,Z 665.469,A -85,B 0,C 180,E1 -6398.495,E2 -6398.495} C_VEL
LIN {X 0,Y 459.346,Z 679.799,A -85,B 0,C 180,E1 -6399.647,E2 -6399.647} C_VEL
LIN {X 0,Y 458.573,Z 692.45,A -85,B 0,C 180,E1 -6400.933,E2 -6400.933} C_VEL
LIN {X 0,Y 457.788,Z 704.66,A -85,B 0,C 180,E1 -6402.497,E2 -6402.497} C_VEL
LIN {X 0,Y 457.187,Z 714.376,A -85,B 0,C 180,E1 -6404.048,E2 -6404.048} C_VEL
LIN {X 0,Y 456.667,Z 723.439,A -85,B 0,C 180,E1 -6405.882,E2 -6405.882} C_VEL
LIN {X 0,Y 456.336,Z 730.507,A -85,B 0,C 180,E1 -6407.73,E2 -6407.73} C_VEL
LIN {X 0,Y 456.125,Z 736.064,A -85,B 0,C 180,E1 -6409.728,E2 -6409.728} C_VEL
LIN {X 0,Y 456.031,Z 739.827,A -85,B 0,C 180,E1 -6411.747,E2 -6411.747} C_VEL
LIN {X 0,Y 455.995,Z 741.824,A -85,B 0,C 180,E1 -6413.884,E2 -6413.884} C_VEL
LIN {X 0,Y 455.995,Z 742.011,A -85,B 0,C 180,E1 -6415.869,E2 -6415.869} C_VEL
LIN {X 0,Y 456.022,Z 740.332,A -85,B 0,C 180,E1 -6417.981,E2 -6417.981} C_VEL
LIN {X 0,Y 456.113,Z 736.959,A -85,B 0,C 180,E1 -6420.014,E2 -6420.014} C_VEL
LIN {X 0,Y 456.296,Z 731.683,A -85,B 0,C 180,E1 -6422.022,E2 -6422.022} C_VEL
LIN {X 0,Y 456.625,Z 724.766,A -85,B 0,C 180,E1 -6423.941,E2 -6423.941} C_VEL
LIN {X 0,Y 457.111,Z 716.113,A -85,B 0,C 180,E1 -6425.756,E2 -6425.756} C_VEL
LIN {X 0,Y 457.756,Z 705.839,A -85,B 0,C 180,E1 -6427.46,E2 -6427.46} C_VEL
LIN {X 0,Y 458.507,Z 694.154,A -85,B 0,C 180,E1 -6428.988,E2 -6428.988} C_VEL
LIN {X 0,Y 459.279,Z 681.898,A -85,B 0,C 180,E1 -6430.281,E2 -6430.281} C_VEL
LIN {X 0,Y 460.074,Z 668.123,A -85,B 0,C 180,E1 -6431.428,E2 -6431.428} C_VEL
LIN {X 0,Y 460.816,Z 653.687,A -85,B 0,C 180,E1 -6432.365,E2 -6432.365} C_VEL
LIN {X 0,Y 461.416,Z 638.184,A -85,B 0,C 180,E1 -6433.108,E2 -6433.108} C_VEL
LIN {X 0,Y 461.845,Z 621.52,A -85,B 0,C 180,E1 -6433.651,E2 -6433.651} C_VEL
LIN {X 0,Y 462.178,Z 592.418,A -85,B 0,C 180,E1 -6434.158,E2 -6434.158} C_VEL
LIN {X 0,Y 463.21,Z 486.346,A -85,B 0,C 180,E1 -6435.85,E2 -6435.85} C_VEL
LIN {X 0,Y 462.002,Z 475.995,A -85,B 0,C 180,E1 -6436.107,E2 -6436.107} C_VEL
LIN {X 0,Y 463.404,Z 432.873,A -85,B 0,C 180,E1 -6439.751,E2 -6439.751} C_VEL
LIN {X 0,Y 464.813,Z 391.796,A -85,B 0,C 180,E1 -6443.195,E2 -6443.195} C_VEL
LIN {X 0,Y 465.885,Z 354.564,A -85,B 0,C 180,E1 -6446.311,E2 -6446.311} C_VEL
LIN {X 0,Y 466.852,Z 313.786,A -85,B 0,C 180,E1 -6449.71,E2 -6449.71} C_VEL
LIN {X 0,Y 466.736,Z 308.144,A -85,B 0,C 180,E1 -6450.198,E2 -6450.198} C_VEL
LIN {X 0,Y 460.194,Z 288.341,A -85,B 0,C 180,E1 -6452.362,E2 -6452.362} C_VEL
LIN {X 0,Y 457.078,Z 279.857,A -85,B 0,C 180,E1 -6453.373,E2 -6453.373} C_VEL
LIN {X 0,Y 457.067,Z 279.55,A -85,B 0,C 180,E1 -6454.749,E2 -6454.749} C_VEL
LIN {X 0,Y 457.08,Z 279.546,A -85,B 0,C 180,E1 -6458.438,E2 -6458.438} C_VEL
LIN {X 0,Y 457.058,Z 279.548,A -85,B 0,C 180,E1 -6462.165,E2 -6462.165} C_VEL
LIN {X 0,Y 457.039,Z 279.553,A -85,B 0,C 180,E1 -6465.816,E2 -6465.816} C_VEL
LIN {X 0,Y 457.037,Z 279.551,A -85,B 0,C 180,E1 -6469.538,E2 -6469.538} C_VEL
LIN {X 0,Y 457.051,Z 279.549,A -85,B 0,C 180,E1 -6473.215,E2 -6473.215} C_VEL
LIN {X 0,Y 457.073,Z 279.551,A -85,B 0,C 180,E1 -6476.865,E2 -6476.865} C_VEL
LIN {X 0,Y 457.081,Z 279.548,A -85,B 0,C 180,E1 -6480.626,E2 -6480.626} C_VEL
LIN {X 0,Y 457.062,Z 279.55,A -85,B 0,C 180,E1 -6484.391,E2 -6484.391} C_VEL
LIN {X 0,Y 457.042,Z 279.552,A -85,B 0,C 180,E1 -6488.048,E2 -6488.048} C_VEL
LIN {X 0,Y 457.04,Z 279.551,A -85,B 0,C 180,E1 -6491.739,E2 -6491.739} C_VEL
LIN {X 0,Y 457.06,Z 279.545,A -85,B 0,C 180,E1 -6495.349,E2 -6495.349} C_VEL
LIN {X 0,Y 457.077,Z 279.547,A -85,B 0,C 180,E1 -6499.022,E2 -6499.022} C_VEL
LIN {X 0,Y 457.082,Z 279.55,A -85,B 0,C 180,E1 -6502.779,E2 -6502.779} C_VEL
LIN {X 0,Y 457.063,Z 279.554,A -85,B 0,C 180,E1 -6506.533,E2 -6506.533} C_VEL
LIN {X 0,Y 457.046,Z 279.549,A -85,B 0,C 180,E1 -6510.064,E2 -6510.064} C_VEL
LIN {X 0,Y 457.051,Z 279.549,A -85,B 0,C 180,E1 -6513.771,E2 -6513.771} C_VEL
LIN {X 0,Y 457.07,Z 279.548,A -85,B 0,C 180,E1 -6517.454,E2 -6517.454} C_VEL
LIN {X 0,Y 457.079,Z 279.549,A -85,B 0,C 180,E1 -6521.196,E2 -6521.196} C_VEL
LIN {X 0,Y 457.073,Z 279.552,A -85,B 0,C 180,E1 -6524.956,E2 -6524.956} C_VEL
LIN {X 0,Y 457.07,Z 279.628,A -85,B 0,C 180,E1 -6528.654,E2 -6528.654} C_VEL
LIN {X 0,Y 457.159,Z 280.08,A -85,B 0,C 180,E1 -6528.859,E2 -6528.859} C_VEL
LIN {X 0,Y 466.829,Z 303.55,A -85,B 0,C 180,E1 -6532.016,E2 -6532.016} C_VEL
LIN {X 0,Y 472.12,Z 317.423,A -85,B 0,C 180,E1 -6533.69,E2 -6533.69} C_VEL
LIN {X 0,Y 473.387,Z 320.574,A -85,B 0,C 180,E1 -6533.871,E2 -6533.871} C_VEL
LIN {X 0,Y 476.224,Z 340.889,A -85,B 0,C 180,E1 -6534.498,E2 -6534.498} C_VEL
LIN {X 0,Y 471.82,Z 539.098,A -85,B 0,C 180,E1 -6537.925,E2 -6537.925} C_VEL
LIN {X 0,Y 470.935,Z 578.935,A -85,B 0,C 180,E1 -6538.633,E2 -6538.633} C_VEL
LIN {X 0,Y 469.987,Z 599.723,A -85,B 0,C 180,E1 -6539.216,E2 -6539.216} C_VEL
LIN {X 0,Y 468.786,Z 620.058,A -85,B 0,C 180,E1 -6540.019,E2 -6540.019} C_VEL
LIN {X 0,Y 467.408,Z 639.187,A -85,B 0,C 180,E1 -6541.002,E2 -6541.002} C_VEL
LIN {X 0,Y 465.933,Z 657.562,A -85,B 0,C 180,E1 -6542.172,E2 -6542.172} C_VEL
LIN {X 0,Y 464.276,Z 676.292,A -85,B 0,C 180,E1 -6543.623,E2 -6543.623} C_VEL
LIN {X 0,Y 462.695,Z 693.408,A -85,B 0,C 180,E1 -6545.216,E2 -6545.216} C_VEL
LIN {X 0,Y 461.202,Z 709.266,A -85,B 0,C 180,E1 -6546.966,E2 -6546.966} C_VEL
LIN {X 0,Y 459.837,Z 723.952,A -85,B 0,C 180,E1 -6548.876,E2 -6548.876} C_VEL
LIN {X 0,Y 458.599,Z 737.959,A -85,B 0,C 180,E1 -6551.045,E2 -6551.045} C_VEL
LIN {X 0,Y 457.644,Z 749.833,A -85,B 0,C 180,E1 -6553.24,E2 -6553.24} C_VEL
LIN {X 0,Y 456.955,Z 759.754,A -85,B 0,C 180,E1 -6555.428,E2 -6555.428} C_VEL
LIN {X 0,Y 456.438,Z 768.846,A -85,B 0,C 180,E1 -6557.862,E2 -6557.862} C_VEL
LIN {X 0,Y 456.143,Z 776.063,A -85,B 0,C 180,E1 -6560.284,E2 -6560.284} C_VEL
LIN {X 0,Y 455.979,Z 781.782,A -85,B 0,C 180,E1 -6562.821,E2 -6562.821} C_VEL
LIN {X 0,Y 455.93,Z 785.491,A -85,B 0,C 180,E1 -6565.221,E2 -6565.221} C_VEL
LIN {X 0,Y 455.918,Z 787.785,A -85,B 0,C 180,E1 -6567.739,E2 -6567.739} C_VEL
LIN {X 0,Y 455.917,Z 788.456,A -85,B 0,C 180,E1 -6570.253,E2 -6570.253} C_VEL
LIN {X 0,Y 455.92,Z 787.476,A -85,B 0,C 180,E1 -6572.767,E2 -6572.767} C_VEL
LIN {X 0,Y 455.931,Z 784.78,A -85,B 0,C 180,E1 -6575.286,E2 -6575.286} C_VEL
LIN {X 0,Y 456.02,Z 780.371,A -85,B 0,C 180,E1 -6577.814,E2 -6577.814} C_VEL
LIN {X 0,Y 456.208,Z 774.127,A -85,B 0,C 180,E1 -6580.355,E2 -6580.355} C_VEL
LIN {X 0,Y 456.546,Z 766.348,A -85,B 0,C 180,E1 -6582.78,E2 -6582.78} C_VEL
LIN {X 0,Y 457.087,Z 757.112,A -85,B 0,C 180,E1 -6585.09,E2 -6585.09} C_VEL
LIN {X 0,Y 457.844,Z 745.898,A -85,B 0,C 180,E1 -6587.382,E2 -6587.382} C_VEL
LIN {X 0,Y 458.789,Z 733.6,A -85,B 0,C 180,E1 -6589.479,E2 -6589.479} C_VEL
LIN {X 0,Y 459.975,Z 719.116,A -85,B 0,C 180,E1 -6591.554,E2 -6591.554} C_VEL
LIN {X 0,Y 461.275,Z 703.592,A -85,B 0,C 180,E1 -6593.423,E2 -6593.423} C_VEL
LIN {X 0,Y 462.631,Z 687.442,A -85,B 0,C 180,E1 -6595.063,E2 -6595.063} C_VEL
LIN {X 0,Y 464.041,Z 669.844,A -85,B 0,C 180,E1 -6596.565,E2 -6596.565} C_VEL
LIN {X 0,Y 465.46,Z 650.552,A -85,B 0,C 180,E1 -6597.924,E2 -6597.924} C_VEL
LIN {X 0,Y 466.817,Z 630.017,A -85,B 0,C 180,E1 -6599.088,E2 -6599.088} C_VEL
LIN {X 0,Y 467.961,Z 609.395,A -85,B 0,C 180,E1 -6599.999,E2 -6599.999} C_VEL
LIN {X 0,Y 468.92,Z 587.704,A -85,B 0,C 180,E1 -6600.705,E2 -6600.705} C_VEL
LIN {X 0,Y 469.574,Z 565.867,A -85,B 0,C 180,E1 -6601.175,E2 -6601.175} C_VEL
LIN {X 0,Y 471.545,Z 459.985,A -85,B 0,C 180,E1 -6602.995,E2 -6602.995} C_VEL
LIN {X 0,Y 474.41,Z 365.404,A -85,B 0,C 180,E1 -6604.818,E2 -6604.818} C_VEL
LIN {X 0,Y 475.268,Z 338.331,A -85,B 0,C 180,E1 -6605.396,E2 -6605.396} C_VEL
LIN {X 0,Y 473.244,Z 320.921,A -85,B 0,C 180,E1 -6606.064,E2 -6606.064} C_VEL
LIN {X 0,Y 473.057,Z 318.848,A -85,B 0,C 180,E1 -6606.287,E2 -6606.287} C_VEL
LIN {X 0,Y 469.658,Z 307.442,A -85,B 0,C 180,E1 -6607.971,E2 -6607.971} C_VEL
LIN {X 0,Y 466.533,Z 299.194,A -85,B 0,C 180,E1 -6609.534,E2 -6609.534} C_VEL
LIN {X 0,Y 463.899,Z 293.142,A -85,B 0,C 180,E1 -6611.03,E2 -6611.03} C_VEL
LIN {X 0,Y 462.143,Z 289.325,A -85,B 0,C 180,E1 -6612.289,E2 -6612.289} C_VEL
LIN {X 0,Y 460.365,Z 286.081,A -85,B 0,C 180,E1 -6614.037,E2 -6614.037} C_VEL
LIN {X 0,Y 459.937,Z 284.857,A -85,B 0,C 180,E1 -6615.224,E2 -6615.224} C_VEL
LIN {X 0,Y 460.05,Z 284.988,A -85,B 0,C 180,E1 -6616.966,E2 -6616.966} C_VEL
LIN {X 0,Y 460.892,Z 287.554,A -85,B 0,C 180,E1 -6618.739,E2 -6618.739} C_VEL
LIN {X 0,Y 462.508,Z 290.241,A -85,B 0,C 180,E1 -6620.055,E2 -6620.055} C_VEL
LIN {X 0,Y 464.521,Z 294.942,A -85,B 0,C 180,E1 -6621.534,E2 -6621.534} C_VEL
